           IF (#ioSystem[#tempIoSystemIndex].device[#tempGeoAddr.STATION].errorState = "DEV_STATE_FAULT")
           THEN
             #ioSystem[#tempIoSystemIndex].device[#tempGeoAddr.STATION].errorState := "DEV_STATE_WAS_FAULT";
           ELSIF (#ioSystem[#tempIoSystemIndex].device[#tempGeoAddr.STATION].errorState = "DEV_STATE_LOST_CON")
           THEN
             #ioSystem[#tempIoSystemIndex].device[#tempGeoAddr.STATION].errorState := "DEV_STATE_WAS_LOST";
           ELSE
             #ioSystem[#tempIoSystemIndex].device[#tempGeoAddr.STATION].errorState := "DEV_STATE_OK";
           END_IF;
         END_IF;

         // check modules pulled  
       ELSIF (#eventClass = #MODULE_PULLED)
       THEN
         #ioSystem[#tempIoSystemIndex].device[#tempGeoAddr.STATION].error := TRUE;
         #ioSystem[#tempIoSystemIndex].device[#tempGeoAddr.STATION].errorState := "DEV_STATE_FAULT";

         #ioSystem[#tempIoSystemIndex].device[#tempGeoAddr.STATION].slot[#tempGeoAddr.SLOT].slotErrorState := TRUE;

       ELSE
         ;
       END_IF;

       // copy diagnosis information to ShowDiag DB
       "CopyToHmiDB"(deviceIndex := UINT_TO_INT(#tempGeoAddr.STATION),
                     plc := #plc,
                     showPlc := #showPlc,
                     ioSystem := #ioSystem[#tempIoSystemIndex],
                     showIoSystem := #showIoSystem[#tempIoSystemIndex]);

       // set flag to update active IO system for HMI
       #showActIoSystem.diagnosisLoaded := TRUE;

     END_IF;

   //=============================================================================
   // evaluate diagnosis information for PLC
   //=============================================================================
   ELSIF (#tempGeoAddr.AREA = #AREA_CENTRAL)
   THEN

     IF (#tempGeoAddr.SLOT <= "MAX_MODULES_LOCAL")
     THEN
       IF (#eventClass = #MODULE_PLUGGED)
       THEN
         IF (#faultId = #MODULE_MATCHES)
           OR (#faultId = #MODULE_OK)
         THEN
           #plc.slot[#tempGeoAddr.SLOT].slotErrorState := FALSE;
         END_IF;

       ELSIF (#eventClass = #MODULE_PULLED)
       THEN
         #plc.slot[#tempGeoAddr.SLOT].slotErrorState := TRUE;
       ELSE
         ;
       END_IF;

       // copy diagnosis information to ShowDiag DB
       "CopyToHmiDB"(deviceIndex := 0,
                     plc := #plc,
                     showPlc := #showPlc,
                     ioSystem := #ioSystem[#tempIoSystemIndex],
                     showIoSystem := #showIoSystem[#tempIoSystemIndex]);

     END_IF;

   ELSE
     ;
   END_IF;
END_FUNCTION

FUNCTION "RackOrStationFailure" : Void   // FC2086, SCL
{ S7_Optimized_Access := 'TRUE' }
VERSION : 0.1
   VAR_INPUT
      laddr : Hw_Io;   // Hardware identifier
      eventClass : Byte;   // Event class
      faultId : Byte;   // Fault identifier
   END_VAR
   VAR_IN_OUT
      plc : "typePlc";   // The diagnostics structure for one PLC
      showPlc : "typeShowPlc";   // The show diagnostics structure for one PLC
      ioSystem : Array[1.."MAX_SYSTEM"] of "typeIoSystem";   // The diagnostics structure for one IO System
      showIoSystem : Array[1.."MAX_SYSTEM"] of "typeShowIoSystem";   // The show diagnostics structure for one IO System
      showActIoSystem : "typeShowActIoSystem";   // The show diagnostics structure for the selected IO System
   END_VAR
   VAR_TEMP
      index : Int;   // index system
      tempSlotIndex : Int;   // Loop index
      tempIoSystemIndex : Int;   // Index for IO System
      tempGeoAddr : GEOADDR;   // Geographical address of the disturbed Module / Device
      tempRetVal : Int;   // Return value of LOG2GEO
      tempRetValModuleStates : Int;   // Return value system function ModuleStates
      tempDeviceModuleStates : Array[0..127] of Bool;   // Storage of the status of all modules in the PN Devices --> State: Problem
      tempLaddr : Hw_Device;   // logical address of the disturbed Module / Device
   END_VAR
   // Ret_Val : return value function
   VAR CONSTANT
      AREA_CENTRAL : UInt := 0;   // Area ID for PLC
      AREA_PROFINET : UInt := 1;   // Area ID for PROFINET IO
      AREA_PROFIBUS : UInt := 2;   // Area ID for PROFIBUS DP
      SLAVE_DEVICE_RET : Byte := 16#38;   // return of a DP slave / IO device
      SLAVE_DEVICE_FAIL : Byte := 16#39;   // Failure of a DP slave / IO device
      DP_SLAVE_FAIL_RET : Byte := 16#C4;   // Failure/return of a DP slave
      IO_DEVICE_FAIL_RET : Byte := 16#CB;   // Failure/return of a PROFINET IO device
      STATE_PROBLEM : USInt := 5;   // Used for instruction DeviceStates, read out all devices with several problems
   END_VAR
BEGIN
   //=============================================================================
   //SIEMENS AG
   //(c)Copyright 2015 All Rights Reserved
   //-----------------------------------------------------------------------------
   //Library: -
   //Tested with: S7-1516-3 PN/DP FW 1.7
   //Engineering: TIA Portal V13 SP1
   //Restrictions: -
   //Requirements: -
   //Functionality: Call Configuration Control function blocks for PLC and devices
   //-----------------------------------------------------------------------------
   //Change log table:
   //Version  Date       Expert in charge Changes applied
   //01.00.00 24.03.2015 Siemens Industry Online Support First released version
   //=============================================================================

   //=============================================================================
   // evaluate event class from Rack error OB
   // and set information to DiagnosticsData DB
   //=============================================================================

   //=============================================================================
   // determine geographic address of faulty device
   //=============================================================================
   #tempRetVal := LOG2GEO(LADDR := #laddr,
                          GEOADDR := #tempGeoAddr);

   //=============================================================================
   // evaluate diagnosis information for devices in an IO system
   //=============================================================================
   IF (#tempGeoAddr.AREA = #AREA_PROFINET)
     OR (#tempGeoAddr.AREA = #AREA_PROFIBUS)
   THEN

     //===========================================================================
     // determine index for IO system
     //===========================================================================
     FOR #index := 1 TO "MAX_SYSTEM" DO
       IF (#ioSystem[#index].ioSystemId = #tempGeoAddr.IOSYSTEM)
       THEN
         #tempIoSystemIndex := #index;
       END_IF;
     END_FOR;

     IF (#tempIoSystemIndex <= "MAX_SYSTEM")
       AND (#tempGeoAddr.STATION <= "MAX_MODULES_DEVICE")
       AND (#tempGeoAddr.SLOT <= "MAX_MODULES_DEVICE")
     THEN
       // check DP slave or IO device return 
       IF (#eventClass = #SLAVE_DEVICE_RET)
       THEN
         // reset error state only if the slave or device state is OK
         IF (#faultId = #DP_SLAVE_FAIL_RET)
           OR (#faultId = #IO_DEVICE_FAIL_RET)
         THEN
           #ioSystem[#tempIoSystemIndex].device[#tempGeoAddr.STATION].error := FALSE;

           FOR #tempSlotIndex := 0 TO #ioSystem[#tempIoSystemIndex].device[#tempGeoAddr.STATION].actualConfiguredModules DO
             #ioSystem[#tempIoSystemIndex].device[#tempGeoAddr.STATION].slot[#tempSlotIndex].slotErrorState := FALSE;
           END_FOR;

           IF (#ioSystem[#tempIoSystemIndex].device[#tempGeoAddr.STATION].errorState = "DEV_STATE_FAULT")
           THEN
             #ioSystem[#tempIoSystemIndex].device[#tempGeoAddr.STATION].errorState := "DEV_STATE_WAS_FAULT";
           ELSIF (#ioSystem[#tempIoSystemIndex].device[#tempGeoAddr.STATION].errorState = "DEV_STATE_LOST_CON")
           THEN
             #ioSystem[#tempIoSystemIndex].device[#tempGeoAddr.STATION].errorState := "DEV_STATE_WAS_LOST";
           ELSE
             #ioSystem[#tempIoSystemIndex].device[#tempGeoAddr.STATION].errorState := "DEV_STATE_OK";
           END_IF;

         ELSE

           // The device is reachable, but faulty because of an error in a
           // subordinated system --> check the modules
           #tempRetVal := GEO2LOG(LADDR => #tempLaddr,
                                  GEOADDR := #tempGeoAddr);

           #tempRetValModuleStates := ModuleStates(LADDR := #tempLaddr,
                                                   MODE := #STATE_PROBLEM,
                                                   STATE := #tempDeviceModuleStates);

           IF (#tempRetValModuleStates = 0)
           THEN
             // Store the state of the different module in the diag DB
             FOR #tempSlotIndex := 0 TO #ioSystem[#tempIoSystemIndex].device[#tempGeoAddr.STATION].actualConfiguredModules DO
               IF (#tempDeviceModuleStates[#tempSlotIndex + 1] = TRUE)
               THEN
                 #ioSystem[#tempIoSystemIndex].device[#tempGeoAddr.STATION].slot[#tempSlotIndex].slotErrorState := TRUE;
               ELSE
                 #ioSystem[#tempIoSystemIndex].device[#tempGeoAddr.STATION].slot[#tempSlotIndex].slotErrorState := FALSE;
               END_IF;
             END_FOR;
           END_IF;

           #ioSystem[#tempIoSystemIndex].device[#tempGeoAddr.STATION].errorState := "DEV_STATE_FAULT";

         END_IF;

         // check DP slave or IO device failure 
       ELSIF (#eventClass = #SLAVE_DEVICE_FAIL)
       THEN
         #ioSystem[#tempIoSystemIndex].device[#tempGeoAddr.STATION].error := TRUE;
         #ioSystem[#tempIoSystemIndex].device[#tempGeoAddr.STATION].errorState := "DEV_STATE_LOST_CON";

         FOR #tempSlotIndex := 0 TO #ioSystem[#tempIoSystemIndex].device[#tempGeoAddr.STATION].actualConfiguredModules DO
           IF #ioSystem[#tempIoSystemIndex].device[#tempGeoAddr.STATION].slot[#tempSlotIndex].slotLaddr <> 0
           THEN
             #ioSystem[#tempIoSystemIndex].device[#tempGeoAddr.STATION].slot[#tempSlotIndex].slotErrorState := TRUE;
           END_IF;
         END_FOR;

       ELSE
         ;
       END_IF;

       // copy diagnosis information to ShowDiag DB
       "CopyToHmiDB"(deviceIndex := UINT_TO_INT(#tempGeoAddr.STATION),
                     plc := #plc,
                     showPlc := #showPlc,
                     ioSystem := #ioSystem[#tempIoSystemIndex],
                     showIoSystem := #showIoSystem[#tempIoSystemIndex]);

       // set flag to update active IO system for HMI
       #showActIoSystem.diagnosisLoaded := TRUE;

     END_IF;

   //=============================================================================
   //evaluate diagnosis information for PLC
   //=============================================================================
   ELSIF (#tempGeoAddr.AREA = #AREA_CENTRAL)
   THEN

     IF (#tempGeoAddr.SLOT <= "MAX_MODULES_LOCAL")
     THEN
       // check DP slave or IO device return 
       IF (#eventClass = #SLAVE_DEVICE_RET)
       THEN
         IF (#faultId = #DP_SLAVE_FAIL_RET)
           OR (#faultId = #IO_DEVICE_FAIL_RET)
         THEN
           #plc.slot[#tempGeoAddr.SLOT].slotErrorState := FALSE;
         END_IF;

         // check DP slave or IO device failure 
       ELSIF (#eventClass = #SLAVE_DEVICE_FAIL)
       THEN
         #plc.slot[#tempGeoAddr.SLOT].slotErrorState := TRUE;
       ELSE
         ;
       END_IF;

       // copy diagnosis information to ShowDiag DB
       "CopyToHmiDB"(deviceIndex := UINT_TO_INT(#tempGeoAddr.STATION),
                     plc := #plc,
                     showPlc := #showPlc,
                     ioSystem := #ioSystem[#tempIoSystemIndex],
                     showIoSystem := #showIoSystem[#tempIoSystemIndex]);

     END_IF;

   ELSE
     ;
   END_IF;
END_FUNCTION

ORGANIZATION_BLOCK "Diagnostic error interrupt"   // OB82, FBD, DiagnosticErrorInterrupt
{ S7_Optimized_Access := 'TRUE' }
VERSION : 0.1
// //============================================================================
// //SIEMENS AG
// //(c)Copyright 2015 All Rights Reserved
// //-----------------------------------------------------------------------------
// //Library: -
// //Tested with: S7-1516-3 PN/DP FW 1.7
// //Engineering: TIA Portal V13 SP1
// //Restrictions: -
// //Requirements: -
// //Functionality: Diagnostic interrupt OB to evaluate diagnosis information for PLC and devices
// //-----------------------------------------------------------------------------
// //Change log table:
// //Version  Date       Expert in charge Changes applied
// //01.00.00 24.03.2015 Siemens Industry Online Support First released version
// //============================================================================
   VAR_INPUT
      IO_State : Word;   // IO state of the HW object
      LADDR : Hw_Any;   // Hardware identifier
      Channel : UInt;   // Channel number
      MultiError : Bool;   // =true if more than one error is present
   END_VAR
BEGIN

REGION Network 1: call function to evaluate diagnosis information
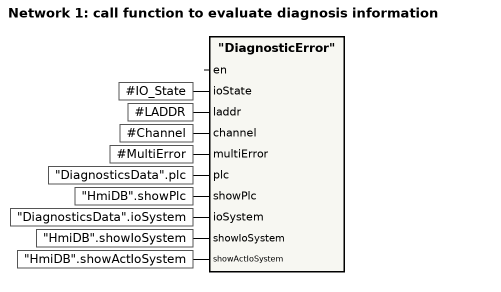
   "DiagnosticError"(ioState := #IO_State,
                     laddr := #LADDR,
                     channel := #Channel,
                     multiError := #MultiError,
                     plc := "DiagnosticsData".plc,
                     showPlc := "HmiDB".showPlc,
                     ioSystem := "DiagnosticsData".ioSystem,
                     showIoSystem := "HmiDB".showIoSystem,
                     showActIoSystem := "HmiDB".showActIoSystem);
END_REGION
END_ORGANIZATION_BLOCK

ORGANIZATION_BLOCK "Pull or plug of modules"   // OB83, FBD, PullPlug
{ S7_Optimized_Access := 'TRUE' }
VERSION : 0.1
// //============================================================================
// //SIEMENS AG
// //(c)Copyright 2015 All Rights Reserved
// //-----------------------------------------------------------------------------
// //Library: -
// //Tested with: S7-1516-3 PN/DP FW 1.7
// //Engineering: TIA Portal V13 SP1
// //Restrictions: -
// //Requirements: -
// //Functionality: Pull/plug interrupt OB to evaluate diagnosis information for PLC and devices
// //-----------------------------------------------------------------------------
// //Change log table:
// //Version  Date       Expert in charge Changes applied
// //01.00.00 24.03.2015 Siemens Industry Online Support First released version
// //============================================================================
   VAR_INPUT
      LADDR : Hw_Io;   // Hardware identifier
      Event_Class : Byte;   // 16#38/39: module inserted, removed
      Fault_ID : Byte;   // Fault identifier
   END_VAR
BEGIN

REGION Network 1: call function to evaluate diagnosis information
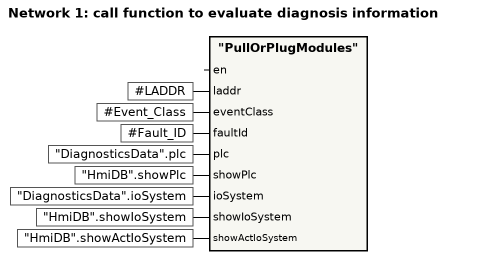
   "PullOrPlugModules"(laddr := #LADDR,
                       eventClass := #Event_Class,
                       faultId := #Fault_ID,
                       plc := "DiagnosticsData".plc,
                       showPlc := "HmiDB".showPlc,
                       ioSystem := "DiagnosticsData".ioSystem,
                       showIoSystem := "HmiDB".showIoSystem,
                       showActIoSystem := "HmiDB".showActIoSystem);
END_REGION
END_ORGANIZATION_BLOCK

ORGANIZATION_BLOCK "Rack or station failure"   // OB86, FBD, RackStationFailure
{ S7_Optimized_Access := 'TRUE' }
VERSION : 0.1
// //============================================================================
// //SIEMENS AG
// //(c)Copyright 2015 All Rights Reserved
// //-----------------------------------------------------------------------------
// //Library: -
// //Tested with: S7-1516-3 PN/DP FW 1.7
// //Engineering: TIA Portal V13 SP1
// //Restrictions: -
// //Requirements: -
// //Functionality: Rack error OB to evaluate diagnosis information for PLC and devices
// //-----------------------------------------------------------------------------
// //Change log table:
// //Version  Date       Expert in charge Changes applied
// //01.00.00 24.03.2015 Siemens Industry Online Support First released version
// //============================================================================
   VAR_INPUT
      LADDR : Hw_Io;   // Hardware identifier
      Event_Class : Byte;   // Event class
      Fault_ID : Byte;   // Fault identifier
   END_VAR
BEGIN

REGION Network 1: call function to evaluate diagnosis information
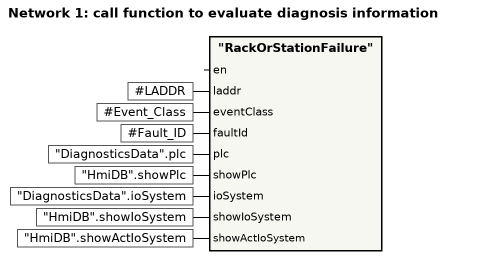
   "RackOrStationFailure"(laddr := #LADDR,
                          eventClass := #Event_Class,
                          faultId := #Fault_ID,
                          plc := "DiagnosticsData".plc,
                          showPlc := "HmiDB".showPlc,
                          ioSystem := "DiagnosticsData".ioSystem,
                          showIoSystem := "HmiDB".showIoSystem,
                          showActIoSystem := "HmiDB".showActIoSystem);
END_REGION
END_ORGANIZATION_BLOCK

ORGANIZATION_BLOCK "MainDiagnostics"   // OB123, FBD, ProgramCycle
TITLE = "Main Program Sweep (Cycle)"
{ S7_Optimized_Access := 'TRUE' }
VERSION : 0.1
// //============================================================================
// //SIEMENS AG
// //(c)Copyright 2015 All Rights Reserved
// //-----------------------------------------------------------------------------
// //Library: -
// //Tested with: S7-1516-3 PN/DP FW 1.7
// //Engineering: TIA Portal V13 SP1
// //Restrictions: -
// //Requirements: -
// //Functionality: Cyclic OB for diagnostics
// //-----------------------------------------------------------------------------
// //Change log table:
// //Version  Date       Expert in charge Changes applied
// //01.00.00 24.03.2015 Siemens Industry Online Support First released version
// //============================================================================
   VAR_INPUT
      Initial_Call : Bool;   // Initial call of this OB
      Remanence : Bool;   // =True, if remanent data are available
   END_VAR
BEGIN

REGION Network 1: call function block Diagnostics
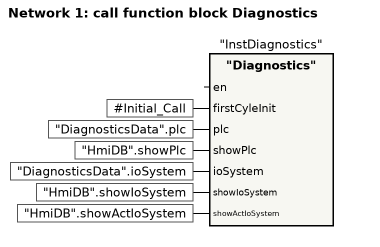
   "InstDiagnostics"(firstCyleInit := #Initial_Call,   // "Diagnostics"
                     plc := "DiagnosticsData".plc,
                     showPlc := "HmiDB".showPlc,
                     ioSystem := "DiagnosticsData".ioSystem,
                     showIoSystem := "HmiDB".showIoSystem,
                     showActIoSystem := "HmiDB".showActIoSystem);
END_REGION
END_ORGANIZATION_BLOCK

// folder: EPICS_Communication

FUNCTION_BLOCK "Tsend_Trecv"   // FB300, SCL
TITLE = TCP1 send receive channel
{ S7_Optimized_Access := 'FALSE' }
AUTHOR : CSL
FAMILY : TSTMP
NAME : S_R_TCP1
VERSION : 1.0
   VAR_INPUT
      INIT_COM : Bool;
      RECV_DB : Variant;
      SEND_DB : Variant;
   END_VAR
   VAR_IN_OUT
      C_PARAM : "CommParam";
   END_VAR
   VAR
      T_SEND : TSEND;
      T_RECV : TRCV;
      T_CONN : TCON;
      T_PARAM : TCON_IP_v4;
      COM1 : Struct
         CONNECTED : Bool;
         CONN_DONE : Bool;
         CONN_BUSY : Bool;
         CONN_ERROR : Bool;
         CONN_STATUS : Word;
         CONN_SETA : Bool;
         SEND_REQ : Bool;
         SEND_DONE : Bool;
         SEND_BUSY : Bool;
         SEND_ERROR : Bool;
         SEND_REQ_P : Bool;
         SEND_STATUS : Word;
         ACT_SEND : Bool;
         RECV_NDR : Bool;
         RECV_BUSY : Bool;
         RECV_ERROR : Bool;
         RECV_STATUS : Word;
         RECV_LEN : UDInt;
      END_STRUCT;
      PLC_COUNT : UDInt;
   END_VAR
   VAR_TEMP
      current_time : Time;
      TMP_PORT : DInt;
   END_VAR
BEGIN

   // Set communication initialisation bit at restart
   #C_PARAM.init_com := #INIT_COM;

   //Clear Bits to start initial connection and communication
   IF #C_PARAM.init_com THEN
       #COM1.CONNECTED := FALSE;
       #COM1.SEND_REQ := FALSE;
       #COM1.CONN_SETA := FALSE;
   END_IF;

   //set TCPx connection parametres 
   #T_PARAM.InterfaceId :=  WORD_TO_UINT (#C_PARAM.interface_id);
   #T_PARAM.ID := #C_PARAM.conn_id;
   #T_PARAM.ConnectionType := #C_PARAM.connection_type;
   #T_PARAM.ActiveEstablished := #C_PARAM.active_established;
   //T_PARAM.RemotePort := 0; 
   #T_PARAM.LocalPort := #C_PARAM.local_port;

   //Establish TCP connection
   //After the connection has been established, it is automatically monitored and maintained by the operating system of the CPU.
   //If the connection has been interrupted, by any line break or due to the remote communications partner, the active partner attempts to reestablish the connection.
   //Therefore, the FB 65 "TCON" may not be called again! 
   IF NOT #COM1.CONNECTED THEN
       #T_CONN(REQ := #COM1.CONN_SETA,
               ID := #C_PARAM.conn_id,
               DONE => #COM1.CONN_DONE,
               BUSY => #COM1.CONN_BUSY,
               ERROR => #COM1.CONN_ERROR,
               STATUS => #COM1.CONN_STATUS,
               CONNECT := #T_PARAM);
   END_IF;

   //Establish connection
   //While startup phase (initial).
   //Indication of the connection status:
   //a) If the CPU may establish the specified connection after Stop/Run immediately, the variable "CONNECTED" indicates HIGH (=1).
   //b) If the CPU is not able to establish the specified connection after Stop/Run, the variable "CONNECTED" remains LOW(=0).
   //c) Note: If the instance DB is loaded by the user, the variable "CONNECTED" indicates HIGH, although the connection may not be established yet. 
   //However, the FB64 "TRCV" would indicate the STATUS=0x80C4, as long as the connection has NOT been established. 
   IF #C_PARAM.init_com THEN
       #COM1.CONN_SETA := TRUE;
   END_IF;
   IF #COM1.CONN_DONE THEN
       #COM1.CONN_SETA := FALSE;
       #C_PARAM.init_com := FALSE;
   END_IF;
   IF #COM1.CONN_SETA THEN
       #COM1.CONNECTED := FALSE;
   ELSE
       #COM1.CONNECTED := TRUE;
   END_IF;

   //generate send trigger pulse
   #current_time := TIME_TCK(); // TIME
   IF (#C_PARAM.sendinterval < ABS(TIME_TO_DINT(#current_time - #C_PARAM.sendtime)) + 1) THEN
       #C_PARAM.sendtrigger := TRUE;
       #C_PARAM.sendtime := #C_PARAM.sendtime + DINT_TO_TIME(#C_PARAM.sendinterval);  //#C_PARAM.sendtime := #current_time;
       #COM1.SEND_REQ_P := FALSE;
   END_IF;

   //Invoke T_SEND function. 
   //IF connection is established TO transmit the data TO the partner as a message.
   // DATA and LEN from input C_PARAM
   IF #COM1.CONNECTED THEN
       #T_SEND(REQ := #COM1.SEND_REQ,
               ID := #C_PARAM.conn_id,
               LEN := #C_PARAM.send_len,
               DONE => #COM1.SEND_DONE,
               BUSY => #COM1.SEND_BUSY,
               ERROR => #COM1.SEND_ERROR,
               STATUS => #COM1.SEND_STATUS,
               DATA := #SEND_DB);//"datatoIOC_TCP1".CommToIOC);
   END_IF;

   //Generate the rising edge SEND_REQ to start the T_SEND function. 
   IF #C_PARAM.sendtrigger AND NOT #COM1.SEND_REQ_P AND NOT #COM1.SEND_BUSY THEN
        #COM1.SEND_REQ := TRUE;
   END_IF;
   #COM1.SEND_REQ_P := #C_PARAM.sendtrigger;

   IF #COM1.SEND_DONE OR #COM1.SEND_ERROR THEN
       #COM1.SEND_REQ := FALSE;
       #C_PARAM.sendtrigger := FALSE;
   END_IF;


   //Invoke T_RECV function
   //The data is stored into the buffer specified with DATA parameter. 
   //After the data has been received, the data is immediately available in the receive buffer. 
   //Receiving is indicated BY the NDR output parameter.
   //Note: DATA and LEN from input C_PARAM 
   IF #COM1.CONNECTED THEN
       #T_RECV(EN_R := #COM1.CONNECTED,
               ID := #C_PARAM.conn_id,
               LEN := #C_PARAM.recv_len,
               ADHOC := false,
               NDR => #COM1.RECV_NDR,
               BUSY => #COM1.RECV_BUSY,
               ERROR => #COM1.RECV_ERROR,
               STATUS => #COM1.RECV_STATUS,
               RCVD_LEN => #COM1.RECV_LEN,
               DATA := #RECV_DB);//"datatoPLC_TCP1".CommToPLC);  

       //Send by request
       //IF (#T_RECV.RCVD_LEN > 0) THEN
       //    #COM1.SEND_REQ := TRUE;
       //END_IF;

   END_IF;
END_FUNCTION_BLOCK

FUNCTION "Send_Receive" : Void   // FC105, SCL
TITLE = Send and receive
{ S7_Optimized_Access := 'FALSE' }
AUTHOR : CSL
FAMILY : TSTMP
NAME : snd_rcv
VERSION : 1.0
BEGIN
   // "channel_param_TCP1".cParam.enable := true;
   //"CH_PARAM_TCP".TCP2_Instance.cParam.enable := true;
   //"CH_PARAM_TCP".TCP3_Instance.cParam.enable := true;
   //

   "TCP1_instance"(INIT_COM := False,
                   RECV_DB := "CPU_WDATA",
                   SEND_DB := "CPU_RDATA",
                   C_PARAM := "CH_PARAM_TCP_CPU".CommParam);     // IN_OUT: STRUCT
   "CPU_Send_RQ":P := "CH_PARAM_TCP_CPU".CommParam.sendtrigger;

   "TCP2_instance"(INIT_COM := False,
                   RECV_DB:="AF_WDATA",
                   SEND_DB:="AF_RDATA",
                   C_PARAM:="CH_PARAM_TCP_AF".CommParam);

   "TCP3_instance"(INIT_COM := False,
                   RECV_DB:="DIO_WDATA",
                   SEND_DB:="DIO_RDATA",
                   C_PARAM:="CH_PARAM_TCP_DIO".CommParam);

   "TCP4_instance"(INIT_COM := False,
                   RECV_DB := "PSU_WDATA",
                   SEND_DB := "PSU_RDATA",
                   C_PARAM := "CH_PARAM_TCP_PSU".CommParam);

   // "TCP4_instance"(INIT_COM := "channel_param_TCP4".cParam.restart,
   //                 C_PARAM := "channel_param_TCP4".cParam,
   //                 DBAnyRecv := "channel_param_TCP4".DBAnyIN,
   //                 DBAnySend := "channel_param_TCP4".DBAnyOUT);
END_FUNCTION

// folder: Gersemi_Communication

FUNCTION "Gersemi_Com" : Void   // FC400, LAD
{ S7_Optimized_Access := 'TRUE' }
VERSION : 0.1
   VAR_TEMP
      stat : Word;   // temporary status
      err : Bool;   // temporary error
   END_VAR
BEGIN

REGION Network 1
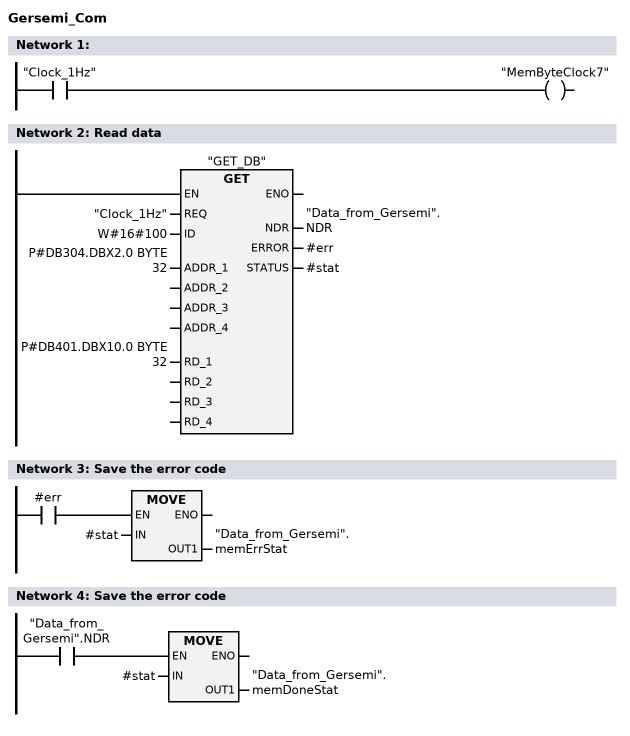
   RUNG wire#powerrail
      Contact( "Clock_1Hz" )
      Coil( "MemByteClock7" )
   END_RUNG
   // the same network as SCL:
   "MemByteClock7" := "Clock_1Hz";
END_REGION

REGION Network 2: Read data
   "GET_DB"(REQ := "Clock_1Hz",   // GET
            ID := W#16#100,
            ADDR_1 := P#DB304.DBX2.0 BYTE 32,
            RD_1 := P#DB401.DBX10.0 BYTE 32,
            NDR => "Data_from_Gersemi".NDR,
            ERROR => #err,
            STATUS => #stat);
END_REGION

REGION Network 3: Save the error code
   RUNG wire#powerrail
      Contact( #err )
      Move(in := #stat, out1 => "Data_from_Gersemi".memErrStat)
   END_RUNG
   // the same network as SCL:
   IF #err THEN "Data_from_Gersemi".memErrStat := #stat; END_IF;
END_REGION

REGION Network 4: Save the error code
   RUNG wire#powerrail
      Contact( "Data_from_Gersemi".NDR )
      Move(in := #stat, out1 => "Data_from_Gersemi".memDoneStat)
   END_RUNG
   // the same network as SCL:
   IF "Data_from_Gersemi".NDR THEN "Data_from_Gersemi".memDoneStat := #stat; END_IF;
END_REGION
END_FUNCTION

// folder: SignalProcessing

FUNCTION "CHKVARS" : Void   // FC9, SCL
TITLE = Check vars
{ S7_Optimized_Access := 'FALSE' }
AUTHOR : ESS_AB
FAMILY : CHKVARS
NAME : AF_CHK
VERSION : 0.1
// This function gets all parameters from the data structure and calls the processing functions
BEGIN

   //Update the actual state and set state to EPICS
   ////"CPU_RDATA".CPU_CONF.ACT_STAT := "mb_actState";
   ////"CPU_RDATA".CPU_CONF.SET_STATE := "mw_setState";

   //IF ("CPU_WDATA".CPU_CONF.WR_DATA) THEN
   "CPU_RDATA".CPU_CONF.TEST_ALL_AD := "CPU_WDATA".CPU_CONF.TEST_ALL_AD;

   IF ("CPU_WDATA".CPU_CONF.OP_MODE <> 0) THEN
       "CPU_RDATA".CPU_CONF.OP_MODE := "CPU_WDATA".CPU_CONF.OP_MODE;
       "CPU_WDATA".CPU_CONF.OP_MODE := 0;
   END_IF;

   "CPU_RDATA".CPU_CONF.OFF := "CPU_WDATA".CPU_CONF.OFF;
   "CPU_RDATA".CPU_CONF.AUX := "CPU_WDATA".CPU_CONF.AUX;
   "CPU_RDATA".CPU_CONF.FIL := "CPU_WDATA".CPU_CONF.FIL;
   "CPU_RDATA".CPU_CONF.STDBY := "CPU_WDATA".CPU_CONF.STDBY;
   "CPU_RDATA".CPU_CONF.HVON := "CPU_WDATA".CPU_CONF.HVON;
   "CPU_RDATA".CPU_CONF.RFON := "CPU_WDATA".CPU_CONF.RFON;
   //"CPU_WDATA".CPU_CONF.RESET := False;
   "CPU_WDATA".CPU_CONF.WR_DATA := FALSE;
   IF ("CPU_WDATA".CPU_CONF.RESET) THEN
       "CPU_RDATA".CPU_CONF.RESET := TRUE;
       "CPU_WDATA".CPU_CONF.RESET := FALSE;
   END_IF;
   //END_IF;

   ////"AD_INTERFACE"(TEST_ALL_AD := "mbi_testAllAds",
   ////               RESET_ALL_AD := "mbi_ResetAllAds",
   ////               CPU_CONF := "CPU_RDATA".CPU_CONF);

   //Copy the RESET_COMMAND into CPU read DB and clear the write command
   //IF ("CPU_RDATA".CPU_CONF.RESET) THEN
       //"CPU_RDATA".CPU_CONF.RESET := "CPU_WDATA".CPU_CONF.RESET;
       //"CPU_WDATA".CPU_CONF.RESET := FALSE;
   //END_IF;

   ////IF ("CPU_RDATA".CPU_CONF.ACK_REQ) THEN
   ////    "mbi_resetledStatus" := "Clock_0.5Hz";
   ////ELSE
   ////    "mbi_resetledStatus" := False;
   ////END_IF;

   //"mbi_resetledStatus" := "CPU_RDATA".CPU_CONF.RESET;

   // IF ("CPU_WDATA".CPU_CONF.SET_STATE <> 0) THEN
   //     "mw_setState" := "CPU_WDATA".CPU_CONF.SET_STATE;
   //     "CPU_RDATA".CPU_CONF.SET_STATE :="CPU_WDATA".CPU_CONF.SET_STATE;
   //     "CPU_WDATA".CPU_CONF.SET_STATE := 0;
   // END_IF;

   //Set new user command from EPICS
   //"mw_setState" := "CPU_WDATA".CPU_CONF.OFF;
   //"CPU_RDATA".CPU_CONF.SET_STATE := "CPU_WDATA".CPU_CONF.OFF;


   //Clear CPU warning bit each cycle
   "CPU_RDATA".CPU_CONF.ACK_REQ := FALSE;

   //Clear CPU force/disable warning bit each check-vars cycle
   "CPU_RDATA".CPU_CONF.FORCE_DIS_MODE_ACT := FALSE;

   //AF_PROCESS gets all information about the data structure and generate the 
   //interlock and warning flags, it also scale the engineering units from the field value.
   //The return value will be stored into the same structure, this information can be watched
   //into the same variable structure.

   //This function gets the CPU_PLC structure, and it contains the information
   //about the operation modes, latched mode, CPU interlock/warning, reset command and
   //some other commands are required to the EPICS communication (See RF-LPS document for more details).

   //Analogue Float signals processing
   //

   "AF_PROCESS"(AFR_STAT := "AF_RDATA".KLY_IP_ISn_Current,             //Analog Float READ type
                AFW_STAT := "AF_WDATA".KLY_IP_ISn_Current,             //Analog Float WRITE type
                CPU_CONF := "CPU_RDATA".CPU_CONF);                     //CPU Data structure type


       "AF_PROCESS"(AFR_STAT := "AF_RDATA".KLY_Oil_TSn_SurfTemp,           //Analog Float READ type
                    AFW_STAT := "AF_WDATA".KLY_Oil_TSn_SurfTemp,           //Analog Float WRITE type
                    CPU_CONF := "CPU_RDATA".CPU_CONF);
       IF (TRUE) THEN
       "AF_PROCESS"(AFR_STAT := "AF_RDATA".KLY_Oil_FSn_WatOutletFlow,      //Analog Float READ type
                    AFW_STAT := "AF_WDATA".KLY_Oil_FSn_WatOutletFlow,      //Analog Float WRITE type
                    CPU_CONF := "CPU_RDATA".CPU_CONF);

       "AF_PROCESS"(AFR_STAT := "AF_RDATA".KLY_Oil_TSn_WatInletTemp,       //Analog Float READ type
                    AFW_STAT := "AF_WDATA".KLY_Oil_TSn_WatInletTemp,       //Analog Float WRITE type
                    CPU_CONF := "CPU_RDATA".CPU_CONF);

       "AF_PROCESS"(AFR_STAT := "AF_RDATA".KLY_Sol_TSn_WatInletTemp,       //Analog Float READ type
                    AFW_STAT := "AF_WDATA".KLY_Sol_TSn_WatInletTemp,       //Analog Float WRITE type
                    CPU_CONF := "CPU_RDATA".CPU_CONF);

       "AF_PROCESS"(AFR_STAT := "AF_RDATA".KLY_Sol_TSn_WatInletTempMan,    //Analog Float READ type
                    AFW_STAT := "AF_WDATA".KLY_Sol_TSn_WatInletTempMan,    //Analog Float WRITE type
                    CPU_CONF := "CPU_RDATA".CPU_CONF);

       "AF_PROCESS"(AFR_STAT := "AF_RDATA".KLY_Sol_TSn_WatOutletTemp,    //Analog Float READ type
                    AFW_STAT := "AF_WDATA".KLY_Sol_TSn_WatOutletTemp,    //Analog Float WRITE type
                    CPU_CONF := "CPU_RDATA".CPU_CONF);

       "AF_PROCESS"(AFR_STAT := "AF_RDATA".KLY_Sol_FSn_WatOutletFlow,      //Analog Float READ type
                    AFW_STAT := "AF_WDATA".KLY_Sol_FSn_WatOutletFlow,      //Analog Float WRITE type
                    CPU_CONF := "CPU_RDATA".CPU_CONF);

       "AF_PROCESS"(AFR_STAT := "AF_RDATA".KLY_Sol_TSn_SurfTemp,           //Analog Float READ type
                    AFW_STAT := "AF_WDATA".KLY_Sol_TSn_SurfTemp,           //Analog Float WRITE type
                    CPU_CONF := "CPU_RDATA".CPU_CONF);

       "AF_PROCESS"(AFR_STAT := "AF_RDATA".KLY_Win_FSn_WatOutletFlow,      //Analog Float READ type
                    AFW_STAT := "AF_WDATA".KLY_Win_FSn_WatOutletFlow,      //Analog Float WRITE type
                    CPU_CONF := "CPU_RDATA".CPU_CONF);

       "AF_PROCESS"(AFR_STAT := "AF_RDATA".KLY_Win_TSn_WatOutletTemp,      //Analog Float READ type
                    AFW_STAT := "AF_WDATA".KLY_Win_TSn_WatOutletTemp,      //Analog Float WRITE type
                    CPU_CONF := "CPU_RDATA".CPU_CONF);

       "AF_PROCESS"(AFR_STAT := "AF_RDATA".KLY_Win_TSn_WatOutletTempMan,   //Analog Float READ type
                    AFW_STAT := "AF_WDATA".KLY_Win_TSn_WatOutletTempMan,   //Analog Float WRITE type
                    CPU_CONF := "CPU_RDATA".CPU_CONF);

       "AF_PROCESS"(AFR_STAT := "AF_RDATA".KLY_Win_TSn_WatOutletSleeveTemp,//Analog Float READ type
                    AFW_STAT := "AF_WDATA".KLY_Win_TSn_WatOutletSleeveTemp,//Analog Float WRITE type
                    CPU_CONF := "CPU_RDATA".CPU_CONF);

       "AF_PROCESS"(AFR_STAT := "AF_RDATA".KLY_Coll_TSn_TopTemp,           //Analog Float READ type
                    AFW_STAT := "AF_WDATA".KLY_Coll_TSn_TopTemp,           //Analog Float WRITE type
                    CPU_CONF := "CPU_RDATA".CPU_CONF);

       "AF_PROCESS"(AFR_STAT := "AF_RDATA".KLY_Coll_TSn_EdgeTemp,          //Analog Float READ type
                    AFW_STAT := "AF_WDATA".KLY_Coll_TSn_EdgeTemp,          //Analog Float WRITE type
                    CPU_CONF := "CPU_RDATA".CPU_CONF);

       "AF_PROCESS"(AFR_STAT := "AF_RDATA".KLY_Coll_TSn_WatInletTemp,      //Analog Float READ type
                    AFW_STAT := "AF_WDATA".KLY_Coll_TSn_WatInletTemp,      //Analog Float WRITE type
                    CPU_CONF := "CPU_RDATA".CPU_CONF);

       "AF_PROCESS"(AFR_STAT := "AF_RDATA".KLY_Coll_TSn_WatOutletTemp,     //Analog Float READ type
                    AFW_STAT := "AF_WDATA".KLY_Coll_TSn_WatOutletTemp,     //Analog Float WRITE type
                    CPU_CONF := "CPU_RDATA".CPU_CONF);

       "AF_PROCESS"(AFR_STAT := "AF_RDATA".KLY_Coll_FSn_WatOutletFlow,     //Analog Float READ type
                    AFW_STAT := "AF_WDATA".KLY_Coll_FSn_WatOutletFlow,     //Analog Float WRITE type
                    CPU_CONF := "CPU_RDATA".CPU_CONF);

       "AF_PROCESS"(AFR_STAT := "AF_RDATA".KLY_Body_TSn_WatInletTemp,      //Analog Float READ type
                    AFW_STAT := "AF_WDATA".KLY_Body_TSn_WatInletTemp,      //Analog Float WRITE type
                    CPU_CONF := "CPU_RDATA".CPU_CONF);

       "AF_PROCESS"(AFR_STAT := "AF_RDATA".KLY_Body_TSn_WatOutletTemp,     //Analog Float READ type
                    AFW_STAT := "AF_WDATA".KLY_Body_TSn_WatOutletTemp,     //Analog Float WRITE type
                    CPU_CONF := "CPU_RDATA".CPU_CONF);

       "AF_PROCESS"(AFR_STAT := "AF_RDATA".KLY_Body_FSn_WatOutletFlow,     //Analog Float READ type
                    AFW_STAT := "AF_WDATA".KLY_Body_FSn_WatOutletFlow,     //Analog Float WRITE type
                    CPU_CONF := "CPU_RDATA".CPU_CONF);

       "AF_PROCESS"(AFR_STAT := "AF_RDATA".KLY_Coll_CollDissipation,       //Analog Float READ type
                    AFW_STAT := "AF_WDATA".KLY_Coll_CollDissipation,       //Analog Float WRITE type
                    CPU_CONF := "CPU_RDATA".CPU_CONF);

       "AF_PROCESS"(AFR_STAT := "AF_RDATA".KLY_Body_BodyDisssipation,      //Analog Float READ type
                    AFW_STAT := "AF_WDATA".KLY_Body_BodyDisssipation,      //Analog Float WRITE type
                    CPU_CONF := "CPU_RDATA".CPU_CONF);

       "AF_PROCESS"(AFR_STAT := "AF_RDATA".RFDS_Circ_FSn_WatOutletFlow,    //Analog Float READ type
                    AFW_STAT := "AF_WDATA".RFDS_Circ_FSn_WatOutletFlow,    //Analog Float WRITE type
                    CPU_CONF := "CPU_RDATA".CPU_CONF);

       "AF_PROCESS"(AFR_STAT := "AF_RDATA".RFDS_Circ_TSn_WatInletTemp,     //Analog Float READ type
                    AFW_STAT := "AF_WDATA".RFDS_Circ_TSn_WatInletTemp,     //Analog Float WRITE type
                    CPU_CONF := "CPU_RDATA".CPU_CONF);

       "AF_PROCESS"(AFR_STAT := "AF_RDATA".RFDS_Load_TSn_WatInletTemp,     //Analog Float READ type
                    AFW_STAT := "AF_WDATA".RFDS_Load_TSn_WatInletTemp,     //Analog Float WRITE type
                    CPU_CONF := "CPU_RDATA".CPU_CONF);

       "AF_PROCESS"(AFR_STAT := "AF_RDATA".RFDS_Load_FSn_WatOutletFlow,     //Analog Float READ type
                    AFW_STAT := "AF_WDATA".RFDS_Load_FSn_WatOutletFlow,     //Analog Float WRITE type
                    CPU_CONF := "CPU_RDATA".CPU_CONF);

       "AF_PROCESS"(AFR_STAT := "AF_RDATA".RFDS_Load_TSn_WatOutletTemp,     //Analog Float READ type
                    AFW_STAT := "AF_WDATA".RFDS_Load_TSn_WatOutletTemp,     //Analog Float WRITE type
                    CPU_CONF := "CPU_RDATA".CPU_CONF);                              //CPU Data structure type
   END_IF;


   // Collector and Body dissipation calculation

   "AF_RDATA".KLY_Coll_CollDissipation.EGU :=
                   ("AF_RDATA".KLY_Coll_TSn_WatOutletTemp.EGU - "AF_RDATA".KLY_Coll_TSn_WatInletTemp.EGU) * "AF_RDATA".KLY_Coll_FSn_WatOutletFlow.EGU;
   "AF_RDATA".KLY_Coll_CollDissipation.EGU :=
                   ("AF_RDATA".KLY_Body_TSn_WatOutletTemp.EGU - "AF_RDATA".KLY_Body_TSn_WatInletTemp.EGU) * "AF_RDATA".KLY_Body_FSn_WatOutletFlow.EGU;
   // Fake data for a test                


   //Digital IO signals processing
                   "DIO_PROCESS"(DIOW_STAT := "DIO_WDATA".EE_1_POWER_PERM,
                                 DIOR_STAT := "DIO_RDATA".EE_1_POWER_PERM,
                                 CPU_CONF := "CPU_RDATA".CPU_CONF);

                   "DIO_PROCESS"(DIOW_STAT := "DIO_WDATA".EE_1_REMOTE,
                                 DIOR_STAT := "DIO_RDATA".EE_1_REMOTE,
                                 CPU_CONF := "CPU_RDATA".CPU_CONF);

                   "DIO_PROCESS"(DIOW_STAT := "DIO_WDATA".EE_1_NO_ERROR_CL,
                                 DIOR_STAT := "DIO_RDATA".EE_1_NO_ERROR_CL,
                                 CPU_CONF := "CPU_RDATA".CPU_CONF);

                   "DIO_PROCESS"(DIOW_STAT := "DIO_WDATA".EE_1_CLOSED,
                                 DIOR_STAT := "DIO_RDATA".EE_1_CLOSED,
                                 CPU_CONF := "CPU_RDATA".CPU_CONF);

                   "DIO_PROCESS"(DIOW_STAT := "DIO_WDATA".EE_1_NO_WARNING,
                                 DIOR_STAT := "DIO_RDATA"."EE_1_NO_WARNING",
                                 CPU_CONF := "CPU_RDATA".CPU_CONF);

                   "DIO_PROCESS"(DIOW_STAT := "DIO_WDATA".EE_1_PC_SPA_OK,
                                 DIOR_STAT := "DIO_RDATA".EE_1_PC_SPA_OK,
                                 CPU_CONF := "CPU_RDATA".CPU_CONF);

                   "DIO_PROCESS"(DIOW_STAT := "DIO_WDATA".PC_1_POWER_Failure,
                                 DIOR_STAT := "DIO_RDATA".PC_1_POWER_Failure,
                                 CPU_CONF := "CPU_RDATA".CPU_CONF);

                   "DIO_PROCESS"(DIOW_STAT := "DIO_WDATA".PC_1_CONNECT,
                                 DIOR_STAT := "DIO_RDATA".PC_1_CONNECT,
                                 CPU_CONF := "CPU_RDATA".CPU_CONF);

                   "DIO_PROCESS"(DIOW_STAT := "DIO_WDATA".PC_1_EXT_OUT,
                                 DIOR_STAT := "DIO_RDATA".PC_1_EXT_OUT,
                                 CPU_CONF := "CPU_RDATA".CPU_CONF);


                   "DIO_PROCESS"(DIOW_STAT := "DIO_WDATA".EB_OK,
                                 DIOR_STAT := "DIO_RDATA".EB_OK,
                                 CPU_CONF := "CPU_RDATA".CPU_CONF);

                   "DIO_PROCESS"(DIOW_STAT := "DIO_WDATA".NO_QUENCH,
                                 DIOR_STAT := "DIO_RDATA".NO_QUENCH,
                                 CPU_CONF := "CPU_RDATA".CPU_CONF);

                   "DIO_PROCESS"(DIOW_STAT := "DIO_WDATA".DAQ_OK,
                                 DIOR_STAT := "DIO_RDATA".DAQ_OK,
                                 CPU_CONF := "CPU_RDATA".CPU_CONF);

                   "DIO_PROCESS"(DIOW_STAT := "DIO_WDATA".EE_2_POWER_PERM,
                                 DIOR_STAT := "DIO_RDATA".EE_2_POWER_PERM,
                                 CPU_CONF := "CPU_RDATA".CPU_CONF);

                   "DIO_PROCESS"(DIOW_STAT := "DIO_WDATA".EE_2_REMOTE,
                                 DIOR_STAT := "DIO_RDATA".EE_2_REMOTE,
                                 CPU_CONF := "CPU_RDATA".CPU_CONF);

                   "DIO_PROCESS"(DIOW_STAT := "DIO_WDATA".EE_2_NO_ERROR_CL,
                                 DIOR_STAT := "DIO_RDATA".EE_2_NO_ERROR_CL,
                                 CPU_CONF := "CPU_RDATA".CPU_CONF);

                   "DIO_PROCESS"(DIOW_STAT := "DIO_WDATA".EE_2_CLOSED,
                                 DIOR_STAT := "DIO_RDATA".EE_2_CLOSED,
                                 CPU_CONF := "CPU_RDATA".CPU_CONF);

                   "DIO_PROCESS"(DIOW_STAT := "DIO_WDATA".EE_2_NO_WARNING,
                                 DIOR_STAT := "DIO_RDATA".EE_2_NO_WARNING,
                                 CPU_CONF := "CPU_RDATA".CPU_CONF);

                   "DIO_PROCESS"(DIOW_STAT := "DIO_WDATA".EE_2_PC_SPA_OK,
                                 DIOR_STAT := "DIO_RDATA".EE_2_PC_SPA_OK,
                                 CPU_CONF := "CPU_RDATA".CPU_CONF);

                   "DIO_PROCESS"(DIOW_STAT := "DIO_WDATA".PC_2_POWER_Failure,
                                 DIOR_STAT := "DIO_RDATA".PC_2_POWER_Failure,
                                 CPU_CONF := "CPU_RDATA".CPU_CONF);

                   "DIO_PROCESS"(DIOW_STAT := "DIO_WDATA".PC_2_CONNECT,
                                 DIOR_STAT := "DIO_RDATA".PC_2_CONNECT,
                                 CPU_CONF := "CPU_RDATA".CPU_CONF);

                   "DIO_PROCESS"(DIOW_STAT := "DIO_WDATA".PC_2_EXT_OUT,
                                 DIOR_STAT := "DIO_RDATA".PC_2_EXT_OUT,
                                 CPU_CONF := "CPU_RDATA".CPU_CONF);


                   "DIO_PROCESS"(DIOW_STAT := "DIO_WDATA".DC24V_AUX_OK,
                                 DIOR_STAT := "DIO_RDATA".DC24V_AUX_OK,
                                 CPU_CONF := "CPU_RDATA".CPU_CONF);

                   "DIO_PROCESS"(DIOW_STAT := "DIO_WDATA".DC24V_PLC_OK,
                                 DIOR_STAT := "DIO_RDATA".DC24V_PLC_OK,
                                 CPU_CONF := "CPU_RDATA".CPU_CONF);


                   "DIO_PROCESS"(DIOW_STAT := "DIO_WDATA".CABLE_POS,
                                 DIOR_STAT := "DIO_RDATA".CABLE_POS,
                                 CPU_CONF := "CPU_RDATA".CPU_CONF);


                   "DIO_PROCESS"(DIOW_STAT := "DIO_WDATA".EE_1_OPEN_RQ,
                                 DIOR_STAT := "DIO_RDATA".EE_1_OPEN_RQ,
                                 CPU_CONF := "CPU_RDATA".CPU_CONF);

                   "DIO_PROCESS"(DIOW_STAT := "DIO_WDATA".CLOSE_EE_1,
                                 DIOR_STAT := "DIO_RDATA".CLOSE_EE_1,
                                 CPU_CONF := "CPU_RDATA".CPU_CONF);

                   "DIO_PROCESS"(DIOW_STAT := "DIO_WDATA".RESET_EE_1,
                                 DIOR_STAT := "DIO_RDATA".RESET_EE_1,
                                 CPU_CONF := "CPU_RDATA".CPU_CONF);

                   "DIO_PROCESS"(DIOW_STAT := "DIO_WDATA".PC_1_PERMIT,
                                 DIOR_STAT := "DIO_RDATA".PC_1_PERMIT,
                                 CPU_CONF := "CPU_RDATA".CPU_CONF);

                   "DIO_PROCESS"(DIOW_STAT := "DIO_WDATA".PC_1_EXT,
                                 DIOR_STAT := "DIO_RDATA".PC_1_EXT,
                                 CPU_CONF := "CPU_RDATA".CPU_CONF);

                   "DIO_PROCESS"(DIOW_STAT := "DIO_WDATA".DIRECT_PA,
                                 DIOR_STAT := "DIO_RDATA".DIRECT_PA,
                                 CPU_CONF := "CPU_RDATA".CPU_CONF);

                   "DIO_PROCESS"(DIOW_STAT := "DIO_WDATA".FLSHBX_HVOLT,
                                 DIOR_STAT := "DIO_RDATA".FLSHBX_HVOLT,
                                 CPU_CONF := "CPU_RDATA".CPU_CONF);

                   "DIO_PROCESS"(DIOW_STAT := "DIO_WDATA".FLSHBX_HCUR,
                                 DIOR_STAT := "DIO_RDATA".FLSHBX_HCUR,
                                 CPU_CONF := "CPU_RDATA".CPU_CONF);

                   "DIO_PROCESS"(DIOW_STAT := "DIO_WDATA".FLSHBX_HE,
                                 DIOR_STAT := "DIO_RDATA".FLSHBX_HE,
                                 CPU_CONF := "CPU_RDATA".CPU_CONF);

                   "DIO_PROCESS"(DIOW_STAT := "DIO_WDATA".EE_2_OPEN_RQ,
                                 DIOR_STAT := "DIO_RDATA".EE_2_OPEN_RQ,
                                 CPU_CONF := "CPU_RDATA".CPU_CONF);

                   "DIO_PROCESS"(DIOW_STAT := "DIO_WDATA".CLOSE_EE_2,
                                 DIOR_STAT := "DIO_RDATA".CLOSE_EE_2,
                                 CPU_CONF := "CPU_RDATA".CPU_CONF);

                   "DIO_PROCESS"(DIOW_STAT := "DIO_WDATA".RESET_EE_2,
                                 DIOR_STAT := "DIO_RDATA".RESET_EE_2,
                                 CPU_CONF := "CPU_RDATA".CPU_CONF);

                   "DIO_PROCESS"(DIOW_STAT := "DIO_WDATA".PC_2_PERMIT,
                                 DIOR_STAT := "DIO_RDATA".PC_2_PERMIT,
                                 CPU_CONF := "CPU_RDATA".CPU_CONF);

                   "DIO_PROCESS"(DIOW_STAT := "DIO_WDATA".PC_2_EXT,
                                 DIOR_STAT := "DIO_RDATA".PC_2_EXT,
                                 CPU_CONF := "CPU_RDATA".CPU_CONF);

                   "DIO_PROCESS"(DIOW_STAT := "DIO_WDATA".LEAD_1_TEMP_OK,
                                 DIOR_STAT := "DIO_RDATA".LEAD_1_TEMP_OK,
                                 CPU_CONF := "CPU_RDATA".CPU_CONF);

                   "DIO_PROCESS"(DIOW_STAT := "DIO_WDATA".LEAD_2_TEMP_OK,
                                 DIOR_STAT := "DIO_RDATA".LEAD_2_TEMP_OK,
                                 CPU_CONF := "CPU_RDATA".CPU_CONF);

                   "DIO_PROCESS"(DIOW_STAT := "DIO_WDATA".LEAD_3_TEMP_OK,
                                 DIOR_STAT := "DIO_RDATA".LEAD_3_TEMP_OK,
                                 CPU_CONF := "CPU_RDATA".CPU_CONF);

                   "DIO_PROCESS"(DIOW_STAT := "DIO_WDATA".LEAD_4_TEMP_OK,
                                 DIOR_STAT := "DIO_RDATA".LEAD_4_TEMP_OK,
                                 CPU_CONF := "CPU_RDATA".CPU_CONF);

                   "DIO_PROCESS"(DIOW_STAT := "DIO_WDATA"."CRYO_1.9K",
                                 DIOR_STAT := "DIO_RDATA"."CRYO_1.9K",
                                 CPU_CONF := "CPU_RDATA".CPU_CONF);

                   "DIO_PROCESS"(DIOW_STAT := "DIO_WDATA"."CRYO_4.5K",
                                 DIOR_STAT := "DIO_RDATA"."CRYO_4.5K",
                                 CPU_CONF := "CPU_RDATA".CPU_CONF);

                   "DIO_PROCESS"(DIOW_STAT := "DIO_WDATA".CRYO_300K_HE,
                                 DIOR_STAT := "DIO_RDATA".CRYO_300K_HE,
                                 CPU_CONF := "CPU_RDATA".CPU_CONF);

                   "DIO_PROCESS"(DIOW_STAT := "DIO_WDATA".CRYO_300K_AIR,
                                 DIOR_STAT := "DIO_RDATA".CRYO_300K_AIR,
                                 CPU_CONF := "CPU_RDATA".CPU_CONF);



                   //"DIO_PROCESS"(DIOW_STAT := "DIO_WDATA".HV_OK_300K_AIR,
                   //              DIOR_STAT := "DIO_RDATA".spare_12,
                   //              CPU_CONF := "CPU_RDATA".CPU_CONF);

                   //"DIO_PROCESS"(DIOW_STAT := "DIO_WDATA".HV_OK_COLD,
                   //              DIOR_STAT := "DIO_RDATA".spare_13,
                   //              CPU_CONF := "CPU_RDATA".CPU_CONF);






   //"PSU_RDATA".SOLENOID1."Real" := "PSU_WDATA".SOLENOID1."Real";

   // Call PSU blocks
   ////"PSU_PROCESS_iDB"();

   //Clear CPU reset bit
   "CPU_RDATA".CPU_CONF.RESET := FALSE;
END_FUNCTION

FUNCTION "AF_PROCESS" : Void   // FC10, SCL
TITLE = AF Satus bit comparison
{ S7_Optimized_Access := 'FALSE' }
AUTHOR : ESS_AB
FAMILY : CHKVARS
NAME : AF_ST
VERSION : 0.1
   VAR_IN_OUT
      AFR_STAT : "AF_RST";
      AFW_STAT : "AF_WST";
      CPU_CONF : "CPU_RCONF";
   END_VAR
   VAR_TEMP
      Akt_Retval : Int;
      Out_Clock_Date : Date_And_Time;
   END_VAR
BEGIN
   // ------------------------------------------------------------------------------
   // 
   //  Title       :   AF_PROCESS
   //  Project     :   
   // -------------------------------------------------------------------------------
   //  File        : 
   //  Author      :   Rafael Montano
   //  Created     :   2015-11-26
   //  Last update :   2016-02-01
   //  Platform    :
   //  Standard    :   SCL
   // -------------------------------------------------------------------------------
   //  Description: This function handles the analog variable types according to the
   //               structure AF_RST and AF_WST described on PLC data types ->
   //               SignalProcessing. Converts the field value into a engineering units
   //               according to the device type DTYP.
   //               The function can also simulate, force, disable and add an offset to 
   //               the original value. All those parameters would be reflected on the 
   //               interlock action since the original value can be replaced or modified.
   //               
   //               InOut parameters:
   //                  @Analog read strucutre type     - AF_RST
   //                  @Analog write strucutre type    - AF_WST
   //                  @CPU read structure type        - CPU_RCONF
   //  
   // -------------------------------------------------------------------------------
   //  Copyright (c) 2016 ESS ERIC
   // -------------------------------------------------------------------------------
   //  Revisions  :
   //  Date        Version     Author          Description
   //  2016-02-01  1.0.0       r. montano      Created
   //  2016-02-05  1.0.1       r. montano      Remove Disable function 
   //                                          The limits are now compared >= instead >
   // -------------------------------------------------------------------------------

   //Copy all parameters from EPICS to the read variable
   //Thresholds and simulation values

   //IF #AFW_STAT.WR_DATA THEN
       #AFR_STAT.HIHI := #AFW_STAT.HIHI;
       #AFR_STAT.HIGH := #AFW_STAT.HIGH;
       #AFR_STAT.LOW := #AFW_STAT.LOW;
       #AFR_STAT.LOLO := #AFW_STAT.LOLO;
       #AFR_STAT.AOFF := #AFW_STAT.AOFF;
       #AFW_STAT.WR_DATA := False;
   //END_IF;

   #AFR_STAT.SVAL := #AFW_STAT.SVAL;

   #AFR_STAT.DISABLE := #AFW_STAT.DISABLE;
   #AFR_STAT.FORCE := #AFW_STAT.FORCE;

   //The variable can be scaled according to the Device Type configuration
   "INT_TO_PHYSICAL"(DTYP := #AFR_STAT.DTYP,
                     VAL := #AFR_STAT.VAL,
                     ERROR => #AFR_STAT.ERR,
                     EGU := #AFR_STAT.EGU);

   //Add the scaled offset to the EGU variable
   #AFR_STAT.EGU := #AFR_STAT.EGU + #AFR_STAT.AOFF;

   //If the variable is properly scaled, can be processed by the function
   //Otherwise an interlock is set to the variable
   IF NOT (#AFR_STAT.ERR = W#16#00) THEN
       #AFR_STAT.INTERLOCK := True;
   END_IF;

   //It was removed by request of RF Group
   IF (#CPU_CONF.OP_MODE = "NORMAL_OPERATION") THEN                  //If the CPU is operating in normal mode
       #AFR_STAT.FORCE := False;                      //The Disable bit has to be set to False
       //#AFR_STAT.DISABLE := False;                      //The Force bit has to be set to False
       //It means is NOT possible TO force nothing in normal operation
   END_IF;
   //End change proposed
   //
   // Since this signal is not longer used, let's keep false
   #AFR_STAT.DISABLE := False;                      //The Force bit has to be set to False

   //IF (NOT #AFR_STAT.DISABLE) THEN                     //Variable is not Disabled

       IF (#AFR_STAT.FORCE) THEN                       //Variable being forced
           #CPU_CONF.FORCE_DIS_MODE_ACT := True;       //Inform to the user that some variable is being forced     
           //Warning - threshold comparison SVAL
           IF (#AFR_STAT.LOW >= #AFR_STAT.SVAL) OR      //Force SVAL value smaller than lower warning
               (#AFR_STAT.HIGH <= #AFR_STAT.SVAL) THEN  //Force value smaller than upper warning
               #AFR_STAT.WARNING := TRUE;              //Set warning bit
           ELSIF (#AFR_STAT.WARNING) THEN              //Reset warning bit if applicable
               IF (NOT #CPU_CONF.LATCH_MODE) OR        //CPU not in larched mode
                   //CPU in latched mode and reset command
                   (#CPU_CONF.RESET AND #CPU_CONF.LATCH_MODE) THEN
                   #AFR_STAT.WARNING := FALSE;         //Set warning bit
              END_IF;
          END_IF;
          //Alarm - threshold comparison SVAL
          IF (#AFR_STAT.LOLO >= #AFR_STAT.SVAL) OR      //Forced SVAL value smaller than lower alarm threshold 
              (#AFR_STAT.HIHI <= #AFR_STAT.SVAL) THEN   //Forced SVAL value greater that upper alarm threshold
              #AFR_STAT.INTERLOCK := True;             //Set Alarm/Interlock bit to the variable
          ELSIF (#AFR_STAT.INTERLOCK) THEN             //Reset Interlock if applicable
              IF NOT #CPU_CONF.LATCH_MODE OR           //CPU is not in latched mode
                  //CPU in latched mode and reset command
                  (#CPU_CONF.RESET AND #CPU_CONF.LATCH_MODE) THEN
                  #AFR_STAT.INTERLOCK := False;        //Reset Interlock bit
                  #AFR_STAT.IsFIRST := False;          //Reset IsFirst bit
              END_IF;
          END_IF;
      ELSE                                             //Variable is not forced
          //Warning - threshold comparison EGU
          IF (#AFR_STAT.LOW >= #AFR_STAT.EGU) OR        //EGU Value smaller than lower warning
               (#AFR_STAT.HIGH <= #AFR_STAT.EGU) THEN   //EGU Value greater than upper warning
               #AFR_STAT.WARNING := True;              //Set warning bit
           ELSIF (#AFR_STAT.WARNING) THEN              //Reset warning bit if applicable
               IF (NOT #CPU_CONF.LATCH_MODE) OR        //CPU not in latched mode
                   //CPU in latched mode and reset command
                   (#CPU_CONF.RESET AND #CPU_CONF.LATCH_MODE) THEN
                   #AFR_STAT.WARNING := False;         //Reset warning bit
                   END_IF;
          END_IF;
          //Alarm - threshold comparison EGU
          IF (#AFR_STAT.LOLO >= #AFR_STAT.EGU) OR       //EGU Value smaller than lower alarm
               (#AFR_STAT.HIHI <= #AFR_STAT.EGU) THEN   //EGU Value greater than upper alarm
               //Update Timestamp if a rising-edge interlock is detected
               IF NOT #AFR_STAT.INTERLOCK THEN
                   #Akt_Retval := RD_LOC_T(OUT => #Out_Clock_Date); //RD_LOC_T is only supported by the CPU-1500
                   #AFR_STAT.TMPST := #Out_Clock_Date; //Update time-stamp variable
               END_IF;
               #AFR_STAT.INTERLOCK := True;            //Set Interlock bit
          ELSE
               IF (#AFR_STAT.INTERLOCK) THEN           //Reset Interlock bit if applicable
                   IF (NOT #CPU_CONF.LATCH_MODE) OR    //CPU is not in latched mode
                       (#CPU_CONF.RESET AND #CPU_CONF.LATCH_MODE) THEN
                       #AFR_STAT.INTERLOCK := False;   //Reset Interlock bit
                       #AFR_STAT.IsFIRST := False;     //Reset IsFirst bit
                   END_IF;
               END_IF;
          END_IF;

       END_IF;

       //Update CPU acknowledge request
       //This bit must be clear at the begining of each cycle and set again within 
       //this function in case any variable is warning or interlock
       IF (#AFR_STAT.WARNING OR                //If variable is in Warning state             
           #AFR_STAT.INTERLOCK) THEN           //If variable is in Interlock state             
           #CPU_CONF.ACK_REQ := True;          //Set the ACK_REQ bit to the CPU status
       END_IF;                                         

   // ELSE //Reset Alarm/Warning bits if the variable is disabled
   //     #AFR_STAT.WARNING := False;             //Reset warning bit
   //     #AFR_STAT.INTERLOCK := False;           //Reset Interlock bit
   //     #AFR_STAT.IsFIRST := False;             //Reset IsFirst bit
   //     #CPU_CONF.FORCE_DIS_MODE_ACT := True;   //Set Force/Disable information bit
   // END_IF;

   //Set isFirst bit
   //Before the Interlock the CPU bit is set, let see which Interlock is activated
   IF NOT #CPU_CONF.INTERLOCK THEN
       IF #AFR_STAT.INTERLOCK THEN       //Interlock
           #AFR_STAT.IsFIRST := True;    //Set IsFirst bit      
       END_IF;
   END_IF;
END_FUNCTION

FUNCTION "DIO_PROCESS" : Void   // FC11, SCL
{ S7_Optimized_Access := 'FALSE' }
VERSION : 0.1
   VAR_IN_OUT
      DIOR_STAT : "DIO_RST";
      DIOW_STAT : "DIO_WST";
      CPU_CONF : "CPU_RCONF";
   END_VAR
   VAR_TEMP
      Akt_Retval : Int;
      Out_Clock_Date : Date_And_Time;
   END_VAR
BEGIN
   // ------------------------------------------------------------------------------
   // 
   //  Title       :   DIO_PROCESS
   //  Project     :   
   // -------------------------------------------------------------------------------
   //  File        : 
   //  Author      :   Rafael Montano
   //  Created     :   2015-11-26
   //  Last update :   2016-02-01
   //  Platform    :
   //  Standard    :   SCL
   // -------------------------------------------------------------------------------
   //  Description: This function handles the digital I/O variable types according to 
   //               the data structure DIO_RST and DIO_WST described on PLC data types ->
   //               SignalProcessing. Gets the field value and process the interlock 
   //               according to the CPU data structure configuration Latched, inverted,
   //               etc.
   //               The function can also simulate, force, disable the original value.
   //               All those parameters would be reflected on the interlock action
   //               since the original value can be replaced or modified.
   //               
   //               InOut parameters:
   //                  @Digital read strucutre type    - DIO_RST
   //                  @Digital write strucutre type   - DIO_WST
   //                  @CPU read structure type        - CPU_RCONF
   //  
   // -------------------------------------------------------------------------------
   //  Copyright (c) 2016 ESS ERIC
   // -------------------------------------------------------------------------------
   //  Revisions  :
   //  Date        Version     Author          Description
   //  2016-02-01  1.0.0       r. montano      Created
   //  2016-02-01  1.0.1       r. montano      Removed Disable function
   // -------------------------------------------------------------------------------

   //Copy all parameters from EPICS to the read variable
   //Disable command, force request and simulation value
   //IF (#DIOW_STAT.WR_DATA) THEN
       #DIOR_STAT.SVAL     := #DIOW_STAT.SVAL;
       #DIOR_STAT.DISABLE  := #DIOW_STAT.DISABLE;
       #DIOR_STAT.FORCE    := #DIOW_STAT.FORCE;
       #DIOW_STAT.WR_DATA  := False;
   //END_IF;

   //IF an event is detected, the value will be passed to the AFR_STAT
   //after that, the input variable, AFW_STAT is cleared.
   // IF (#DIOW_STAT.STAT <> FALSE) THEN
   //     //Before set the bits, the program will not allow to change internal bits
   //     #DIO_STAT_BIT[3] := #DIOW_STAT_BIT[3];
   //     #DIO_STAT_BIT[4] := #DIOW_STAT_BIT[4];
   //     #DIOW_STAT.STAT := 0;
   // END_IF;
   // 
   //It was removed by request of RF Group
   IF (#CPU_CONF.OP_MODE = "NORMAL_OPERATION") THEN                  //If the CPU is operating in normal mode
       #DIOR_STAT.FORCE := False;                      //The Disable bit has to be set to False
       //#DIOR_STAT.DISABLE := False;                      //The Force bit has to be set to False
       //It means is NOT possible TO force nothing in normal operation
   END_IF;

   // Since this signal is no longer used, let's keep it false
   #DIOR_STAT.DISABLE := False;                            //The Force bit has to be set to False

   IF #DIOR_STAT.DTYP = "DI" THEN                          //IF digital input variable
       //IF NOT #DIOR_STAT.DISABLE THEN                    //Variable is not disabled
           IF #DIOR_STAT.FORCE THEN                        //Variable is being forced
               #CPU_CONF.FORCE_DIS_MODE_ACT := True;       //Inform to the user that some variable is being forced
               IF #DIOR_STAT.SVAL THEN
                   #DIOR_STAT.INTERLOCK := True;           //Set alarm/interlock bit of variable
                   #CPU_CONF.ACK_REQ := True;              //Set CPU warning bit. This bit must be reset at the begining of each cycle 
                   IF NOT #CPU_CONF.INTERLOCK THEN         //Before the interlock bit of the CPU is set, lets see which interlock is active
                       IF #DIOR_STAT.INTERLOCK THEN        //Interlock
                           #DIOR_STAT.IsFIRST := True;     //Set isFirst bit
                       END_IF;
                   END_IF;
               ELSIF NOT #DIOR_STAT.SVAL THEN              //Force to OFF
                   IF NOT #CPU_CONF.LATCH_MODE OR          //CPU is not latched mode
                       #DIOR_STAT.N_LATCH OR               //NEVERLATCHED Variable
                       (#CPU_CONF.RESET AND #CPU_CONF.LATCH_MODE) THEN //CPU reset command AND latched mode
                           #DIOR_STAT.INTERLOCK := False;  //Clear alarm/interlock bit
                           #DIOR_STAT.IsFIRST := False;    //Clear isFirst bit
                   END_IF;
               END_IF;
           ELSE
               IF #DIOR_STAT.INVERT    AND
                   NOT #DIOR_STAT.VAL   THEN                //Bit invert ON
                       IF NOT #DIOR_STAT.INTERLOCK THEN
                           #Akt_Retval := RD_LOC_T(OUT => #Out_Clock_Date);
                           #DIOR_STAT.TMPST := #Out_Clock_Date;
                       END_IF;
                       #DIOR_STAT.INTERLOCK := True;
                       #CPU_CONF.ACK_REQ := True;           //SET the warning bit in the CPU status.
               ELSIF NOT #DIOR_STAT.INVERT AND
                  #DIOR_STAT.VAL       THEN
                       IF NOT #DIOR_STAT.INTERLOCK THEN
                           #Akt_Retval := RD_LOC_T(OUT => #Out_Clock_Date);
                           #DIOR_STAT.TMPST := #Out_Clock_Date;
                       END_IF;
                       #DIOR_STAT.INTERLOCK := True;
                       #CPU_CONF.ACK_REQ := True;           //SET the warning bit in the CPU status.

               // IF #DIOR_STAT.VAL THEN                      //Variable NOT forced
               //     //There was not interlock detected - Set the timestamp
               //     IF NOT #DIOR_STAT.INTERLOCK THEN
               //         #Akt_Retval := RD_LOC_T(OUT => #Out_Clock_Date);
               //         #DIOR_STAT.TMPST := #Out_Clock_Date;
               //     END_IF;
               //     #DIOR_STAT.INTERLOCK := True;           //Set alarm/interlock bit
               //     #CPU_CONF.ACK_REQ := True;              //SET the warning bit in the CPU status.
               //                                             //This bit must be reset at the begining of each cycle
               //     IF NOT #CPU_CONF.INTERLOCK THEN         //Before the interlock bit of the CPU is set, lets see which intelock is active
               //         IF #DIOR_STAT.INTERLOCK THEN        //Interlock
               //             #DIOR_STAT.IsFIRST := True;     //Set isFirst bit
               //         END_IF;
               //     END_IF;
               ELSIF (#DIOR_STAT.INTERLOCK) THEN            //Clear interlock/alarm bit if applicable
                   IF NOT #CPU_CONF.LATCH_MODE OR           //CPU not in latched mode          
                       #DIOR_STAT.N_LATCH OR                //NEVERLATCHED variable
                       //CPU reset command AND in latched mode
                       (#CPU_CONF.RESET AND #CPU_CONF.LATCH_MODE) THEN
                           #DIOR_STAT.INTERLOCK := False;   //Clear interlock bit
                           #DIOR_STAT.IsFIRST := False;     //Clear isFirst bit
                   ELSIF #CPU_CONF.INTERLOCK THEN           //PLC CPU is not in interlock
                           #CPU_CONF.ACK_REQ := True;       //Keep warning bit in the CPU status.
                                                            //This bit must be reset at the begining of each cycle
                   END_IF;
               END_IF;
           END_IF;
       // ELSE
       //     #DIOR_STAT.INTERLOCK := False;                  //Clear interlock bit
       //     #DIOR_STAT.IsFIRST := False;                    //Clear isFirst bit
       //     #CPU_CONF.FORCE_DIS_MODE_ACT := True;           //Set Force/Disable information bit
       // END_IF;

   ELSIF #DIOR_STAT.DTYP = "DO" THEN                       //If digital output variable
       IF #DIOR_STAT.FORCE THEN                            //Variable being forced
           #CPU_CONF.FORCE_DIS_MODE_ACT := True;           //Inform to the user that some variable is being forced
           #DIOR_STAT.VAL := #DIOR_STAT.SVAL;              //Forced the same value as SVAL
           IF (#DIOR_STAT.INVERT AND                    //Bit invertedDO on
               NOT #DIOR_STAT.VAL) OR                      //Forced to FALSE - INVERTED
               (#DIOR_STAT.INVERT AND                   //Bit invertDO OFF
                   #DIOR_STAT.VAL) THEN                    //Force to TRUE - NOT INVERTED
                   #DIOR_STAT.IsFIRST := True;             //Set isFirst bit
           ELSE
                   #DIOR_STAT.IsFIRST := False;            //Clear isFirst bit
           END_IF;

       ELSE                                                //Variable not forced
           IF #DIOR_STAT.INTERLOCK THEN                    //Alarm/Interlock Output ON
               //Set isFirst
               IF NOT #CPU_CONF.INTERLOCK THEN             //Before the Interlock bit of the CPU is set
                                                           //lets see which interlock is active
                   IF #DIOR_STAT.INTERLOCK THEN
                       #DIOR_STAT.IsFIRST := True;         //Set isFisrt bit
                   END_IF;
               END_IF;

               IF #DIOR_STAT.INVERT THEN                   //Bit invert ON
                   //If an Interlock is not detected before, set the RTC time
                   IF #DIOR_STAT.VAL THEN
                       #Akt_Retval := RD_LOC_T(OUT => #Out_Clock_Date);
                       #DIOR_STAT.TMPST := #Out_Clock_Date;
                   END_IF;
                   #DIOR_STAT.VAL := False;
               ELSE                                        //Bit invert OFF
                   IF NOT #DIOR_STAT.VAL THEN
                       #Akt_Retval := RD_LOC_T(OUT => #Out_Clock_Date);
                       #DIOR_STAT.TMPST := #Out_Clock_Date;
                   END_IF;
                   #DIOR_STAT.VAL := True;
               END_IF;
           ELSE  //Clear alarm bit, latching conditioning are not applicable to OUTPUTS
               #DIOR_STAT.IsFIRST := False;                //Clear isFirst bit            
               IF #DIOR_STAT.INVERT THEN                //Bit invertDO ON
                   #DIOR_STAT.VAL := True;                 //Clear alarm variable by setting OUTPUT
               ELSE
                   #DIOR_STAT.VAL := False;                //Clear alarm variable by resetting OUTPUT
               END_IF;
           END_IF;
       END_IF;
   ELSE
       //If the device type is not defined into the DB, the interlock will be activated to avoid 
       //unallocated variables.
       #DIOR_STAT.INTERLOCK := True;
       #DIOR_STAT.VAL := True;
   END_IF;

   // (*PASS THE ACTUAL VALUE OF THE DIGITAL INPUT/OUTPUT TO THE BIT 0 OF THE STATUS WORD*)
   // IF #DIOR_STAT.VAL THEN (*INPUT/OUPUT ON*)
   //     #DIOR_STAT.VAL := True;   //Reset bit 0 OF status Word, equal TO .VAL
   // ELSE (*INPUT/OUPUT OFF*)
   //     #DIOR_STAT.VAL := False; //Reset bit 0 OF status Word, equal TO .VALE
   // END_IF;
END_FUNCTION

FUNCTION "AD_INTERFACE" : Void   // FC15, SCL
TITLE = Arc detectors interface
{ S7_Optimized_Access := 'FALSE' }
VERSION : 0.1
   VAR_IN_OUT
      CPU_CONF : "CPU_RCONF";
      TEST_ALL_AD : Bool;
      RESET_ALL_AD : Bool;
   END_VAR
   VAR CONSTANT
      PulseDuration : Time := T#1S;
   END_VAR
BEGIN

   // ------------------------------------------------------------------------------
   // 
   //  Title       :   AD_INTERFACE
   //  Project     :   
   // -------------------------------------------------------------------------------
   //  File        : 
   //  Author      :   Rafael Montano
   //  Created     :   2016-07-08
   //  Last update :   2016-07-08
   //  Platform    :
   //  Standard    :   SCL
   // -------------------------------------------------------------------------------
   //  Description: This function handles the command from EPICS regarding the arc 
   //               detector interface. Time Pulse (TP): The function generates a pulse
   //               according to the contant PulseDuraction to test/reset the arc-detectors
   //               unit.
   //                              __|--PulseDuration--|___
   //               InOut parameters:
   //                  @CPU reset command
   //                  @Test all arc detectors output
   //                  @Reset all arc detectors output
   //  
   // -------------------------------------------------------------------------------
   //  Copyright (c) 2016 ESS AB
   // -------------------------------------------------------------------------------
   //  Revisions  :
   //  Date        Version     Author          Description
   //  2016-08-07  1.0         r. montano      Created
   // -------------------------------------------------------------------------------

   "T_ResetAllAD_DB".TP(IN := #CPU_CONF.RESET,
                        PT := #PulseDuration,
                        Q => #RESET_ALL_AD);

   "T_TestAllAD_DB".TP(IN := #CPU_CONF.TEST_ALL_AD,
                       PT := #PulseDuration,
                       Q => #TEST_ALL_AD);
END_FUNCTION

FUNCTION "INT_TO_PHYSICAL" : Void   // FC20, SCL
TITLE = Scale measurement
{ S7_Optimized_Access := 'FALSE' }
AUTHOR : ESS_AB
VERSION : 0.1
// This function scales the field value into an engineering units.
   VAR_INPUT
      DTYP : Byte;
      VAL : Int;
   END_VAR
   VAR_OUTPUT
      ERROR : Word;
   END_VAR
   VAR_IN_OUT
      EGU : Real;
   END_VAR
   VAR_TEMP
      INT_TO_PHYSICAL : Real;
   END_VAR
BEGIN

   // #ERROR code*
   // (W#16#...)      Meaning

   // 0000     ->     No error
   // 0008     ->     The value of the IN parameter is greater than the value of the high limit (HI_LIM) or less than the value of the low limit (LO_LIM).
   // 8XYY     ->     FOR more information on errors, refer TO "See also".
   //     *The error codes can be displayed as integer OR hexadecimal value in the program editor. FOR additional information on toggling display formats, refer TO "See also".


   IF
       #DTYP = "TSn_PT100" THEN
       #EGU := INT_TO_REAL(#VAL) / 10;
       #ERROR := W#16#00;
   ELSIF #DTYP = "TSn_TC" THEN
       #EGU := INT_TO_REAL(#VAL) / 10;
       #ERROR := W#16#00;
   ELSIF #DTYP = "ISn_IP" THEN
       //#INT_TO_PHYSICAL := INT_TO_REAL(#VAL) * 10.0 / 27648.0; (*basic convertion to VOLTS*)
       //#EGU := #INT_TO_PHYSICAL * 10.0; //Temporarily
       #ERROR := SCALE(IN := #VAL,
                       HI_LIM := 100.0,
                       LO_LIM := 0,
                       BIPOLAR := 0,
                       OUT => #EGU);
       #ERROR := W#16#00;
   ELSIF #DTYP = "VSn_0_10v" THEN    //Convert to 0..10V
       #INT_TO_PHYSICAL := INT_TO_REAL(#VAL) * 10.0 / 27648.0; (*basic convertion to VOLTS*)
       #EGU := #INT_TO_PHYSICAL; //Temporarily
       #ERROR := W#16#00;
   ELSIF #DTYP = "FSn_05_80_l_min" THEN
       #INT_TO_PHYSICAL := INT_TO_REAL(#VAL) * 16.0 / 27648.0 + 4.0; (*basic convertion to mAMPS*)
       //The EGU linearisation should be defined with the sensor
       #EGU := (((79.5 / REAL#16.0) * (#INT_TO_PHYSICAL - 4.0))) + 0.5; (*0.5 l/m TO 80 l/m*)
       #ERROR := W#16#00;
   ELSIF #DTYP = "FSn_8_1000_l_min" THEN
       #INT_TO_PHYSICAL := INT_TO_REAL(#VAL) * 16.0 / 27648.0 + 4.0; (*basic convertion to mAMPS*)
       //The EGU linearisation should be defined with the sensor
       #EGU := (((992.0 / REAL#16.0) * (#INT_TO_PHYSICAL - 4.0))) + 8.0; (*8 l/m TO 1000 l/m*)
       #ERROR := W#16#00;
   ELSIF #DTYP = "PSn_0_10_bar" THEN
       #INT_TO_PHYSICAL := INT_TO_REAL(#VAL) * 16.0 / 27648.0 + 4.0; (*basic convertion to mAMPS*)
       #EGU := ((10.0 / REAL#16.0) * (#INT_TO_PHYSICAL - 4.0)); (*0 bar TO 10 bar*)
       #ERROR := W#16#00;
   ELSIF #DTYP = "TSn_0_50_C" THEN
       #INT_TO_PHYSICAL := INT_TO_REAL(#VAL) * 16.0 / 27648.0 + 4.0; (*basic convertion to mAMPS*)
       #EGU := ((50.0 / REAL#16.0) * (#INT_TO_PHYSICAL - 4.0)); (*0 C to 50 C*)
       #ERROR := W#16#00;
   ELSIF #DTYP = "COLL_DISP" THEN
       //Nothing to be done here, the calcullation should be made in CHKVARS function
       #ERROR := W#16#00;
   ELSIF #DTYP = "BODY_DISP" THEN
       //Nothing to be done here, the calcullation should be made in CHKVARS function
       #ERROR := W#16#00;
   ELSIF #DTYP = "ENG_0-30A" THEN
       #ERROR := SCALE(IN := #VAL,
                       HI_LIM := 30,
                       LO_LIM := 0,
                       BIPOLAR := 0,
                       OUT => #EGU);
       #ERROR := W#16#00;
   ELSIF #DTYP = "ENG_0-17A" THEN
       #ERROR := SCALE(IN := #VAL,
                       HI_LIM := 17,
                       LO_LIM := 0,
                       BIPOLAR := 0,
                       OUT => #EGU);
       #ERROR := W#16#00;
   ELSIF #DTYP = "ENG_0-900W" THEN
       #ERROR := SCALE(IN := #VAL,
                       HI_LIM := 900,
                       LO_LIM := 0,
                       BIPOLAR := 0,
                       OUT => #EGU);
       #ERROR := W#16#00;
   ELSIF #DTYP = "ENG_0-300V" THEN
       #ERROR := SCALE(IN := #VAL,
                       HI_LIM := 300,
                       LO_LIM := 0,
                       BIPOLAR := 0,
                       OUT => #EGU);
       #ERROR := W#16#00;
   ELSIF #DTYP = "ISn_0_20mA" THEN
       #ERROR := SCALE(IN := #VAL,
                       HI_LIM := 20.0,
                       LO_LIM := 0.0,
                       BIPOLAR := 0,
                       OUT => #EGU);
   ELSIF #DTYP = "ISn_4_20mA" THEN
       #ERROR := SCALE(IN := #VAL,
                       HI_LIM := 20.0,
                       LO_LIM := 4.0,
                       BIPOLAR := 0,
                       OUT => #EGU);
   ELSIF #DTYP = "ISn_bipolar_20mA" THEN
       #ERROR := SCALE(IN := #VAL,
                       HI_LIM := 20.0,
                       LO_LIM := -20.0,
                       BIPOLAR := 0,
                       OUT => #EGU);
   ELSIF #DTYP = "VSn_bipolar_50mV" THEN
       #ERROR := SCALE(IN := #VAL,
                       HI_LIM := 0.05,
                       LO_LIM := -0.05,
                       BIPOLAR := 1,
                       OUT => #EGU);
   ELSIF #DTYP = "VSn_bipolar_500mV" THEN
       #ERROR := SCALE(IN := #VAL,
                       HI_LIM := 0.5,
                       LO_LIM := -0.5,
                       BIPOLAR := 1,
                       OUT => #EGU);
   ELSIF #DTYP = "VSn_bipolar_1V" THEN
       #ERROR := SCALE(IN := #VAL,
                       HI_LIM := 1,
                       LO_LIM := -1,
                       BIPOLAR := 1,
                       OUT => #EGU);
   ELSIF #DTYP = "NO_CONVERSION" THEN
       #ERROR := W#16#0;
   ELSE
       #EGU := 0.0;
       #ERROR := W#16#10;
   END_IF;
END_FUNCTION

FUNCTION "TD_TO_INT" : Void   // FC50, SCL
{ S7_Optimized_Access := 'FALSE' }
AUTHOR : Rafael
VERSION : 0.1
   VAR_TEMP
      Out_Clock_Date : Date_And_Time;
      Akt_Retval : Int;
      Out_Date : Date;
      Out_Clock : Time_Of_Day;
      temp_day : Int;
   END_VAR
BEGIN
   #Akt_Retval := RD_SYS_T(OUT => #Out_Clock_Date);
   "DateTime".Out_Clock_Date := #Out_Clock_Date;
   "DateTime".Out_Date := DT_TO_DATE(#Out_Clock_Date);
   "DateTime".Out_Time := DT_TO_TOD(#Out_Clock_Date);

   #Akt_Retval := RD_LOC_T(OUT => #Out_Clock_Date);
   "DateTime".Out_Clock_Date_Local := #Out_Clock_Date;
END_FUNCTION

// ===== library types =====

FUNCTION "PHYSICAL_TO_INT" : Void   // FC31, SCL
{ S7_Optimized_Access := 'FALSE' }
VERSION : 0.1
   VAR_INPUT
      DTYP : Byte;
      EGU : Real;
   END_VAR
   VAR_OUTPUT
      VAL : Int;
      ERROR : Word;
   END_VAR
   VAR_TEMP
      TEMP_VALUE : Real;
   END_VAR
BEGIN

   // #ERROR code*
   // (W#16#...)      Meaning

   // 0000     ->     No error
   // 0008     ->     The value of the IN parameter is greater than the value of the high limit (HI_LIM) or less than the value of the low limit (LO_LIM).
   // 8XYY     ->     FOR more information on errors, refer TO "See also".
   //     *The error codes can be displayed as integer OR hexadecimal value in the program editor. FOR additional information on toggling display formats, refer TO "See also".


   IF #DTYP = "TSn" THEN
       #VAL := REAL_TO_INT(#EGU / 100) ;
       #ERROR := W#16#00;
   ELSIF #DTYP = "ENG_0-30A" THEN    //Convert to 0..30A
       #ERROR := UNSCALE(BIPOLAR := 0,
                         HI_LIM :=30.0,
                         IN := #EGU,
                         LO_LIM := 0.0,
                         OUT => #VAL);
   ELSIF #DTYP = "ENG_0-17A" THEN    //Convert to 0..30A
       #ERROR := UNSCALE(BIPOLAR := 0,
                         HI_LIM := 17.0,
                         IN := #EGU,
                         LO_LIM := 0.0,
                         OUT => #VAL);
   ELSE
       #VAL := 0;
       #ERROR := W#16#10;
   END_IF;
END_FUNCTION

// folder: MachineState

FUNCTION "GET_LOCATION" : Void   // FC13, STL
TITLE = Get location
{ S7_Optimized_Access := 'FALSE' }
VERSION : 0.1
   VAR_OUTPUT
      LOCATION : Int;
   END_VAR
   VAR CONSTANT
      LOCAL : Byte := 16#0;
      REMOTE : Byte := 16#1;
   END_VAR
BEGIN

REGION Network 1
   //      A
   //      JC    LOC
   //      L     #LOCAL
   //      T     #LOCATION
   //      BEU
   //
   //LOC:  L     #REMOTE
   //      T     #LOCATION
   //      BEU
   //
   //
END_REGION
END_FUNCTION

FUNCTION "SET_AMP_STATE" : Void   // FC14, STL
TITLE = Set amplifier State
{ S7_Optimized_Access := 'FALSE' }
VERSION : 0.1
   VAR_IN_OUT
      CPU_CONF : "CPU_RCONF";
      SET_STATE : Int;
   END_VAR
BEGIN

REGION Network 1: Set new command to the target 0=OFF; 1=AUX; 2=FIL; 3=STDBY; 4=HVON; 5=RFON
         A     "mbi_resetCmd";
         JC    RESET;

         A     "mbi_offCmd";
         O     #CPU_CONF.OFF;
   //      FP    "mbi_swPulseOff"
         JC    OFF;

         A     "mbi_auxCmd";
         O     #CPU_CONF.AUX;
         JC    AUX;

         A     "mbi_filCmd";
         O     #CPU_CONF.FIL;
         JC    FIL;

         A     "mbi_stdbyCmd";
         O     #CPU_CONF.STDBY;
         JC    STDBY;

         A     "mbi_hvonCmd";
         O     #CPU_CONF.HVON;
         JC    HVON;

         A     "mbi_rfonCmd";
         O     #CPU_CONF.RFON;
         JC    RFON;
         BEU;

   OFF:  L     "OFF";
         T     #SET_STATE;
         R     #CPU_CONF.OFF;
         BEU;

   AUX:  L     "AUX";
         T     #SET_STATE;
         R     #CPU_CONF.AUX;
         BEU;

   FIL:  L     "FIL";
         T     #SET_STATE;
         R     #CPU_CONF.FIL;
         BEU;

   STDBY:L     "STDBY";
         T     #SET_STATE;
         R     #CPU_CONF.STDBY;
         BEU;

   HVON: L     "HVON";
         T     #SET_STATE;
         R     #CPU_CONF.HVON;
         BEU;

   RFON: L     "RFON";
         T     #SET_STATE;
         R     #CPU_CONF.RFON;
         BEU;

   RESET:S     #CPU_CONF.RESET;
   //     R     #CPU_CONF.RESET
END_REGION
END_FUNCTION

FUNCTION "STATE_FAULTS" : Void   // FC21, STL
{ S7_Optimized_Access := 'FALSE' }
VERSION : 0.1
   VAR_TEMP
      T_MISS_COND : Byte;
      STATE : Byte;
      FAULT_STATE : Byte;
   END_VAR
BEGIN

REGION Network 1
   //AUX
         L     "AUX";
         AN    "mbi_auxPre";
         JC    PRE;
         AN    "mbi_auxSup";
         JC    SUP;
   //FIL
         L     "FIL";
         AN    "mbi_filPre";
         JC    PRE;
         AN    "mbi_filSup";
         JC    SUP;
   //STBY
         L     "STDBY";
         AN    "mbi_stbyPre";
         JC    PRE;
         AN    "mbi_stbySup";
         JC    SUP;
   //HVON
         L     "HVON";
         AN    "mbi_hvonPre";
         JC    PRE;
         AN    "mbi_hvonSup";
         JC    SUP;
   //RFON
         L     "RFON";
         AN    "mbi_rfonPre";
         JC    PRE;
         AN    "mbi_rfonSup";
         JC    SUP;

   PRE:  T     #FAULT_STATE;
         JU    REST;

   SUP:  T     #FAULT_STATE;
         JU    REST;

   REST: L     #FAULT_STATE;
         L     2;
         -I;
         T     "mw_setState";
END_REGION
END_FUNCTION

// folder: PowerSupply

FUNCTION_BLOCK "FILAMENT_LOGIC"   // FB3001, SCL
TITLE = Filament logic
{ S7_Optimized_Access := 'FALSE' }
FAMILY : PSU
VERSION : 1.1
// Filament control logic for the Power Supply Unit
   VAR_INPUT
      PSU_TYPE : Int;   // Power Supply Type ID
   END_VAR
   VAR_IN_OUT
      PSU_Outputs : "PSU_Outputs";   // General Output Signals from the PLC to the PSU
      PSU_Inputs : "PSU_Inputs";   // General Input Signals from the PSU to the PLC
      PSU_RSTAT : "FILAMENT_RST";   // PSU Status interface
      CPU_RCONF : "CPU_RCONF";   // SIM_GlobalData_Read
      CPU_WCONF : "CPU_WCONF";   // SIM_GlobalData_Write
      START_CMD : Bool;   // Start Command for StateMachine
      STOP_CMD : Bool;   // Stop Command for StateMachine
      PSU_WSTAT : "FILAMENT_WST";
   END_VAR
   VAR
      ERROR_STAT : Word;   // Internal variable for ERROR bits
      ERRORS AT ERROR_STAT : Array[0..15] of Bool;   // Internal variable for ERROR bits
      DeviceCooled : TON_TIME;   // After turning off the PSU the time till the device gets cold
      BlindOut : TON_TIME;   // Blind out Limit checking
      PSU_UptimeNoHV : TON_TIME;   // Uptime timer in secs
      StaysWarm : Time;   // After a proper PSU run, how long can a warm start to be triggered
      MaxCurrentForFilament : Real;   // The Maximum current for the filament defined by the supplier
      MaxPowerForFilament : Real;   // The Maximum Power for the filament defined by the supplier
      MaxCurrentForSolenoid : Real;   // The Maximum current for the filament defined by the supplier
      MaxVoltageForSolenoid : Real;   // The Maximum Power for the filament defined by the supplier
      AlarmBlindOutTime : Time;   // After turning on the PSU, the time till the limits supervisions are disabled
      BlindOut_DONE : Bool;   // Limits can be monitored now
      TEMP_IPGM : Real;   // Temp Current Output
      TEMP_IMON : Real;   // Temp Curernt Input
      TEMP_WMON : Real;   // Temp Power Input
      TEMP_VMON : Real;   // Temp Voltage Input
      SP1_Length : DInt;   // SP1 Timer length (100ms)
      SP2_Length : DInt;   // SP2 Timer length (100ms)
      SP3_Length : DInt;   // SP3 Timer length (100ms)
      TEMP_ACTUAL_SETPOINT : Int;   // Actual SetPoint
      TEMP_PSU_ON : Bool;   // Temp variable for PSU_ON
      TEMP_PSU_STARTED : Bool;   // Temp variable for PSU_STARTED
      TEMP_PSU_STOPPED : Bool;   // Temp variable for PSU_STOPPED
      TEMP_PSU_RESET : Bool;   // Temp variable for PSU_RESET
      TEMP_PSU_WARMUP : Bool;   // Temp variable for PSU_WARMUP
      TEMP_PSU_TEMP_REACHED : Bool;   // Temp variable for PSU_TEMP_REACHED
      SP1_WarmUpTime_TICK : Bool;   // SP1 Timer tick
      SP2_WarmUpTime_TICK : Bool;   // SP2 Timer tick
      SP3_WarmUpTime_TICK : Bool;   // SP3 Timer tick
      DeviceCooled_TICK : Bool;   // After PSU is stopped, the device got cold
      UptimeNoHV_TICK : Bool;   // Timer Tick bit
      V_SCALE_ERROR : Word;   // Scaling Error
      I_SCALE_ERROR : Word;   // Scaling Error
      W_SCALE_ERROR : Word;   // Scaling Error
      SP1_WarmupTimer : TON_TIME;
      SP2_WarmupTimer : TON_TIME;
      SP3_WarmupTimer : TON_TIME;
      SP1_CurrTime : Time;
      SP2_CurrTime : Time;
      SP3_CurrTime : Time;
      WARMUP_MONITOR_CurrTime : Time;
      WarmupMonitor_Tick : Bool;
      TEMP_Interlock : Bool;
      TEMP_Warning : Bool;
      TEMP_InterlockNeeded : Bool;
      TEMP_WarningNeeded : Bool;
      PSU_STARTCMD_TP : TP_TIME;
      PSU_STARTCMD_TICK : Bool;
      PSU_RESETCMD_TP : TP_TIME;
      PSU_RESETCMD_TICK : Bool;
      PSU_STOPCMD_TP : TP_TIME;
      PSU_STOPCMD_TICK : Bool;
      PSU_STARTCMD_TP_WIRED : TP_TIME;
      PSU_STARTCMD_TICK_WIRED : Bool;
      PSU_STOPCMD_TP_WIRED : TP_TIME;
      PSU_STOPCMD_TICK_WIRED : Bool;
      TEMP_CurrentRampRate : Real;
      IPGM_BeforeInterlock : Real;
      WARMUP_MONITOR : TON_TIME;
      TimeStampUpdated : Bool;
      Temp_Tol_Warmup : Real;
   END_VAR
   VAR_TEMP
      ReadCLK_retval : Int;
   END_VAR
BEGIN
   //Description: This FILAMENT_LOGIC FB handles all Filament related tasks.
   //Author: Miklos Boros Tel:+36702072273 email:borosmiklos@gmail.com
   //Last update: 2016.12.05 11:00
   //Version: v1.0
   //Change log at the bottom of the code!

   //Error Bits description ***************************

           //Bit0;   EpicsBit8:  Initialisation error. No DTYP is given!
           //Bit1;   EpicsBit9:  PSU is in LOCAL mode. Set to REMOTE!
           //Bit2;   EpicsBit10: Analog Input IMON SCALE error!
           //Bit3;   EpicsBit11: Analog Input WMON SCALE error!
           //Bit4;   EpicsBit12: Analog Input VMON SCALE error!
           //Bit5;   EpicsBit13: Analog OutPut IPGM/VPGM SCALE error!
           //Bit6;   EpicsBit14: SP1 Current value can't be zero if Ramped!
           //Bit7;   EpicsBit15: SP2 Current value can't be zero if Ramped!
           //Bit8;   EpicsBit0:  SP3 Current value can't be zero if Ramped!
           //Bit9;   EpicsBit1:  PSU SetPoint values are not in incresing order!
           //Bit10;  EpicsBit2:  Interlock PSU has internal faliure!
           //Bit11;  EpicsBit3:  Interlock during Warmup! 
           //Bit12;  EpicsBit4:  Interlock absulute maximum exeeded!
           //Bit13;  EpicsBit5:  Interlock High limit exeeded while PSU_ON!
           //Bit14;  EpicsBit6:  Interlock Low limit exeeded while PSU_ON!
           //Bit15;  EpicsBit7:  PSU can't be turned on because of an error!

           //IF (#PSU_WSTAT.WR_DATA) THEN

           // If the total warmup time if minor than 2.0, then the set the 
           // value to 2.0 as a minumum set-point
           IF (#PSU_WSTAT.TOL_InWARMUP_SP < 2.0) THEN
               #PSU_WSTAT.TOL_InWARMUP_SP := 2.0;
               #Temp_Tol_Warmup := #PSU_WSTAT.TOL_InWARMUP_SP;
           ELSE
               #Temp_Tol_Warmup := #PSU_WSTAT.TOL_InWARMUP_SP;
           END_IF;

               //Feedback EPICS commands
               #PSU_RSTAT.I_RAMP_ON := #PSU_WSTAT.I_RAMP_ON;
               #PSU_RSTAT.V_RAMP_ON := #PSU_WSTAT.V_RAMP_ON;
               #PSU_RSTAT.FORCE_ON := #PSU_WSTAT.FORCE;
               #PSU_RSTAT.TOL_InWARMUP := #Temp_Tol_Warmup;

               //Feedback Low Limits for Current and Power  !Note: the high alarm and warnings are Filament Type specific because of the Max allowed current and power
               #PSU_RSTAT.I_LOLO := #PSU_WSTAT.I_LOLO;
               #PSU_RSTAT.I_LOW := #PSU_WSTAT.I_LOW;
               #PSU_RSTAT.W_LOLO := #PSU_WSTAT.W_LOLO;
               #PSU_RSTAT.W_LOW := #PSU_WSTAT.W_LOW;

               IF (NOT #TEMP_PSU_WARMUP) THEN //Setpoint can be changed from HMI only when it's not warming up
                   #PSU_RSTAT.TIME_COLD_SP1 := #PSU_WSTAT.TIME_COLD_SP1;
                   #PSU_RSTAT.TIME_WARM_SP1 := #PSU_WSTAT.TIME_WARM_SP1;
                   #PSU_RSTAT.I_SP1 := #PSU_WSTAT.I_SP1;

                   #PSU_RSTAT.TIME_COLD_SP2 := #PSU_WSTAT.TIME_COLD_SP2;
                   #PSU_RSTAT.TIME_WARM_SP2 := #PSU_WSTAT.TIME_WARM_SP2;
                   #PSU_RSTAT.I_SP2 := #PSU_WSTAT.I_SP2;

                   #PSU_RSTAT.TIME_COLD_SP3 := #PSU_WSTAT.TIME_COLD_SP3;
                   #PSU_RSTAT.TIME_WARM_SP3 := #PSU_WSTAT.TIME_WARM_SP3;
                   #PSU_RSTAT.I_SP3 := #PSU_WSTAT.I_SP3;
               END_IF;

               //FORCE INPUT SIGNALS **************************
               //Feedback SIMULATION values
               #PSU_RSTAT.S_FAULT := #PSU_WSTAT.S_FAULT;
               #PSU_RSTAT.S_I_REG := #PSU_WSTAT.S_IVAL;
               #PSU_RSTAT.S_LOC_REM := #PSU_WSTAT.S_LOC_REM;
               #PSU_RSTAT.S_ON_STATUS := #PSU_WSTAT.S_ON_STATUS;
               #PSU_RSTAT.S_IMON := #PSU_WSTAT.S_IMON;
               #PSU_RSTAT.S_WMON := #PSU_WSTAT.S_WMON;

               IF (#PSU_RSTAT.FORCE_ON) THEN // If the FORCE in the HMI is pressed
                   IF (#PSU_RSTAT.N_FORCE = FALSE) THEN //Simulation of the values if NFORCE allows it
                       //Take all the Simulated values from EPICS
                       #PSU_Inputs.LOC_REM := #PSU_WSTAT.S_LOC_REM;
                       #PSU_Inputs.I_REG := #PSU_WSTAT.S_IVAL;
                       #PSU_Inputs.FAULT := #PSU_WSTAT.S_FAULT;
                       #PSU_Inputs.ON_STATUS := #PSU_WSTAT.S_ON_STATUS;
                       #PSU_RSTAT.IMON := #PSU_WSTAT.S_IMON;
                       #TEMP_IMON := #PSU_WSTAT.S_IMON;
                       #PSU_RSTAT.WMON := #PSU_WSTAT.S_WMON;
                       #TEMP_WMON := #PSU_WSTAT.S_WMON;
                   END_IF;
               END_IF;

               //Feedback the Intelock High limits with check
               IF (#PSU_WSTAT.I_HIHI < #MaxCurrentForFilament) THEN
                   #PSU_RSTAT.I_HIHI := #PSU_WSTAT.I_HIHI;
               ELSE
                   #PSU_RSTAT.I_HIHI := #MaxCurrentForFilament;
               END_IF;
               IF (#PSU_WSTAT.I_HIGH < #MaxCurrentForFilament) THEN
                   #PSU_RSTAT.I_HIGH := #PSU_WSTAT.I_HIGH;
               ELSE
                   #PSU_RSTAT.I_HIGH := #MaxCurrentForFilament;
               END_IF;
               IF (#PSU_WSTAT.W_HIHI < #MaxPowerForFilament) THEN
                   #PSU_RSTAT.W_HIHI := #PSU_WSTAT.W_HIHI;
               ELSE
                   #PSU_RSTAT.W_HIHI := #MaxPowerForFilament;
               END_IF;
               IF (#PSU_WSTAT.W_HIGH < #MaxPowerForFilament) THEN
                   #PSU_RSTAT.W_HIGH := #PSU_WSTAT.W_HIGH;
               ELSE
                   #PSU_RSTAT.W_HIGH := #MaxPowerForFilament;
               END_IF;

               //Feedback the SP1 SP2 SP3 currents with check
               IF (#PSU_WSTAT.I_SP1 < #MaxCurrentForFilament) THEN
                   #PSU_RSTAT.I_SP1 := #PSU_WSTAT.I_SP1;
               ELSE
                   #PSU_RSTAT.I_SP1 := #MaxCurrentForFilament;
               END_IF;
               IF (#PSU_WSTAT.I_SP2 < #MaxCurrentForFilament) THEN
                   #PSU_RSTAT.I_SP2 := #PSU_WSTAT.I_SP2;
               ELSE
                   #PSU_RSTAT.I_SP2 := #MaxCurrentForFilament;
               END_IF;
               IF (#PSU_WSTAT.I_SP3 < #MaxCurrentForFilament) THEN
                   #PSU_RSTAT.I_SP3 := #PSU_WSTAT.I_SP3;
               ELSE
                   #PSU_RSTAT.I_SP3 := #MaxCurrentForFilament;
               END_IF;

               #PSU_WSTAT.WR_DATA := FALSE;
           //END_IF;


           //Init variables
           IF (NOT #TEMP_Interlock) THEN
               #ERROR_STAT := W#0; // Keep the value if an Iterlock happens
           END_IF;
           #TEMP_IPGM := 0.0;


           //First PLC Cícle
           IF (NOT #TEMP_PSU_STARTED) AND (NOT #TEMP_PSU_STOPPED) THEN
               #TEMP_PSU_STOPPED := TRUE;
           END_IF;

           //   WARMUP_T can't be Zero
           IF (#PSU_RSTAT.TOTAL_WARMPUP_T = S5T#0s) THEN
               //Total warmp time (SP1+SP2+SP3) to EPICS
               #PSU_RSTAT.TOTAL_WARMPUP_T := "INT_S5TIME"(((REAL_TO_INT(#PSU_RSTAT.TIME_COLD_SP1) + REAL_TO_INT(#PSU_RSTAT.TIME_COLD_SP2) + REAL_TO_INT(#PSU_RSTAT.TIME_COLD_SP3)) * 10) + 100);
               //#PSU_RSTAT.TOTAL_WARMPUP_T := "INT_S5TIME"(REAL_TO_INT(#PSU_RSTAT.TIME_COLD_SP1) + REAL_TO_INT(#PSU_RSTAT.TIME_COLD_SP2) + REAL_TO_INT(#PSU_RSTAT.TIME_COLD_SP3) + 100);
               IF (#PSU_RSTAT.TOTAL_WARMPUP_T = S5T#0s) THEN
                   #PSU_RSTAT.TOTAL_WARMPUP_T := S5T#60s;
               END_IF;
           END_IF;

           // Warmup tolareace can't be Zero!
           IF (#Temp_Tol_Warmup = 0.0) THEN
               #Temp_Tol_Warmup := 5.0;
           END_IF;




           //COMMON PSU FUNCTIONS **********************
           //FEEDBACK SIGNALS **************************

           //Copy LOC_REM and I_REG to the Read area. These status signals are not calculated they are coming from the PSU.
           #PSU_RSTAT.LOC_REM_ST := #PSU_Inputs.LOC_REM;
           #PSU_RSTAT.I_REG := #PSU_Inputs.I_REG;

           IF (#PSU_RSTAT.FORCE_ON) THEN // If the FORCE in the HMI is pressed
               IF (#PSU_RSTAT.N_FORCE = FALSE) THEN //Simulation of the values if NFORCE allows it

                   //Take all the Simulated values from EPICS
                   //#PSU_Inputs.LOC_REM   :=  #PSU_WSTAT.S_LOC_REM;
                   //#PSU_Inputs.I_REG     :=  #PSU_WSTAT.S_IVAL;
                   //#PSU_Inputs.FAULT     :=  #PSU_WSTAT.S_FAULT;
                   //#PSU_Inputs.ON_STATUS :=  #PSU_WSTAT.S_ON_STATUS;
                   //#PSU_RSTAT.IMON       :=  #PSU_WSTAT.S_IMON;
                   //#TEMP_IMON            :=  #PSU_WSTAT.S_IMON;
                   //#PSU_RSTAT.WMON       :=  #PSU_WSTAT.S_WMON;
                   //#TEMP_WMON            :=  #PSU_WSTAT.S_WMON;
                   #CPU_RCONF.FORCE_DIS_MODE_ACT := TRUE;
               END_IF;
           END_IF;

           IF (NOT #PSU_RSTAT.FORCE_ON) OR (#PSU_RSTAT.N_FORCE = TRUE) THEN  //If PSU_FORCE is not applied, or disabled = normal operation

               //Scale IMON 
               "INT_TO_PHYSICAL"(DTYP := "ENG_0-30A",
                                 VAL := #PSU_Inputs.IMON,
                                 EGU => #TEMP_IMON,
                                 ERROR => #I_SCALE_ERROR);
               IF (#I_SCALE_ERROR <> W#0) THEN
                   #ERRORS[2] := TRUE; //PSU IMON SCALE Error
               END_IF;
               #PSU_RSTAT.IMON := #TEMP_IMON;


               //Scale WMON
               "INT_TO_PHYSICAL"(DTYP := "ENG_0-900W",
                                 VAL := #PSU_Inputs.WMON,
                                 EGU => #TEMP_WMON,
                                 ERROR => #W_SCALE_ERROR);
               IF (#W_SCALE_ERROR <> W#0) THEN
                   #ERRORS[3] := TRUE; //PSU WMON SCALE Error
               END_IF;
               #PSU_RSTAT.WMON := #TEMP_WMON;

           END_IF;

           // PSU START COMMAND
           // If the PSU block receives the Start CMD the PSU_STARTED will be SET
           //#PSU_STARTCMD_TP(IN := (#PSU_WSTAT.START), //Pulse generation for START_CMD coming from EPICS 
           //                 PT := t#2s,
           //                 Q => #PSU_STARTCMD_TICK);
           #PSU_STARTCMD_TP_WIRED(IN := (#START_CMD),       //Pulse generation for START_CMD coming from StateMachine
                                  PT := t#2s,
                                  Q => #PSU_STARTCMD_TICK_WIRED);
           IF (#PSU_STARTCMD_TICK OR #PSU_STARTCMD_TICK_WIRED) AND (NOT #TEMP_Interlock) THEN
               #TEMP_PSU_STARTED := TRUE;
               #TEMP_PSU_STOPPED := FALSE;
           END_IF;
           IF (NOT #PSU_STARTCMD_TICK_WIRED) AND #START_CMD THEN
               #START_CMD := FALSE;
           END_IF;

           //PSU Reset COMMAND 
           #TEMP_PSU_RESET := FALSE; // the command is for 2s
           //#PSU_RESETCMD_TP(IN := (#PSU_WSTAT.RESET OR #CPU_RCONF.RESET),
           #PSU_RESETCMD_TP(IN := #CPU_RCONF.RESET,
                            PT := t#2s,
                            Q => #PSU_RESETCMD_TICK);

           IF (#PSU_RESETCMD_TICK) THEN
               #TEMP_PSU_RESET   := TRUE;
           END_IF;

           //#PSU_STOPCMD_TP(IN := (#PSU_WSTAT.STOP), //Pulse generation for STOP_CMD coming from EPICS
           //                PT := t#2s,
           //                Q => #PSU_STOPCMD_TICK);

           #PSU_STOPCMD_TP_WIRED(IN := (#STOP_CMD),       //Pulse generation for STOP_CMD coming from StateMachine
                                 PT := t#2s,
                                 Q => #PSU_STOPCMD_TICK_WIRED);

           //PSU STOP COMMAND 
           IF (#PSU_STOPCMD_TICK OR #PSU_STOPCMD_TICK_WIRED) THEN
               #TEMP_PSU_STOPPED := TRUE;
               #TEMP_PSU_ON := FALSE;
               #TEMP_PSU_STARTED := FALSE;
               #TEMP_PSU_WARMUP := FALSE;
               #TEMP_ACTUAL_SETPOINT := 0;
               #PSU_RSTAT.TOTAL_WARMUP_LEFT := 0;
               #PSU_RSTAT.UPTIME_NO_HV := 0;
               #PSU_RSTAT.WARMUP_LEFT_SP := 0;
               #TEMP_CurrentRampRate := 0.0;
           END_IF;
           IF (NOT #PSU_STOPCMD_TICK_WIRED) AND #STOP_CMD THEN
               #STOP_CMD := FALSE;
           END_IF;

           //PSU TYPE SPECIFIC FUNCTIONS **********************

           IF (#PSU_TYPE = "PSU_NOT_DEFINED") THEN
               //Parametrization ERROR Type_Not_Filled_Out
               #ERRORS[0] := TRUE;
               #TEMP_PSU_STOPPED := TRUE;
               #TEMP_PSU_STARTED := FALSE;
               #TEMP_PSU_ON := FALSE;
               #TEMP_PSU_WARMUP := FALSE;
               #TEMP_ACTUAL_SETPOINT := 0;
               #PSU_RSTAT.TOTAL_WARMUP_LEFT := 0;
               #PSU_RSTAT.UPTIME_NO_HV := 0;
               #PSU_RSTAT.WARMUP_LEFT_SP := 0;
               #TEMP_CurrentRampRate := 0.0;
           END_IF;
           IF (#PSU_TYPE = "PSU_KLYSTRON_FILAMENT") THEN //Type:Klystron FILAMENT Heater

               //Klystron heater TIME constans        
               #StaysWarm := t#5s; //The time till the Filament cools down
               #AlarmBlindOutTime := t#2s; //Time after SP3 is reached (PSU_ON) and Interlock Low checking is enabled
               #MaxCurrentForFilament := 26.0; //Supplier specified Maximum Current (in Amp) 
               #MaxPowerForFilament := 800.0;//Supplier specified Maximum Power (in Watt) 

               //Voltage monitoring is not available for the FILAMENT Heater
               #PSU_RSTAT.VMON := 0.0;


               //Check when the PSU cools down TOF
               #DeviceCooled(IN := NOT #PSU_RSTAT.ON_STATUS,
                             PT := #StaysWarm,
                             Q => #DeviceCooled_TICK);
               IF #DeviceCooled_TICK THEN
                   IF (#TEMP_PSU_TEMP_REACHED = TRUE) AND (NOT #TEMP_PSU_WARMUP) THEN //If the Filament was already warm and not warming up, start all over.
                       #TEMP_ACTUAL_SETPOINT := 0;
                   END_IF;
                   #TEMP_PSU_TEMP_REACHED := FALSE; //The next start can be only a cold start           
               END_IF;


